// TwinCAT 3 PLC project HAWino
// ProgramVersion: 3.1.4024.12
// libraries:
//   Tc2_Standard, * (Beckhoff Automation GmbH)
//   Tc2_System, * (Beckhoff Automation GmbH)
//   Tc2_Utilities, * (Beckhoff Automation GmbH)
//   Tc3_IotBase, * (Beckhoff Automation GmbH)
//   Tc3_JsonXml, * (Beckhoff Automation GmbH)
//   Tc3_Module, * (Beckhoff Automation GmbH)
// project tree:
//   / ControlTask.TcTTO, Kollisionserkennung_1.TcTTO, MQTT_1.TcTTO, PlcTask.TcTTO
//   DUTs/ Auftrag.TcDUT, ControllerState.TcDUT, CoreDriveState.TcDUT, CoreGripperControlState.TcDUT, RobotInternalData.TcDUT, RobotPoseSimple.TcDUT, RobotStatusGW1.TcDUT, U_IpAdr.TcDUT, RobotPose.TcDUT
//   DUTs/PowerManagement/ FleetManagement.TcDUT, ST_PwrMgmt_HAWino.TcDUT, ST_PwrMgmt_HAWino_In.TcDUT, ST_PwrMgmt_HAWino_Out.TcDUT
//   DUTs/Sys/ DUT_SysState.TcDUT
//   GVLs/ ControlParameters.TcGVL, Var_HAWIno.TcGVL
//   POUs/HAWinoCore/ Camera.TcPOU, CameraConnectionUDP.TcPOU, Gripper.TcPOU, IrDistanceFromRaw.TcPOU, IrDistanceSensors.TcPOU, MotorDrivers.TcPOU, MQTT.TcPOU, PowerManager.TcPOU, WheelEncoders.TcPOU, HAWino.TcPOU
//   POUs/UserPOUs/GW2/ AStar.TcPOU, DS_GW1.TcPOU, Fahrauftrag.TcPOU, Kollisionserkennung.TcPOU, ReadAssigment.TcPOU
//   POUs/UserPOUs/GW3ControlAlgorithm/ CollisionDetector.TcPOU, KalmanObserver.TcPOU, NonLinearController.TcPOU, Robot.TcPOU, SimpleObserver.TcPOU, PController.TcPOU, SimpleTrajectory.TcPOU, TimeOptimalTrajectory.TcPOU, ControlPRG.TcPOU, VelocityMeasurement.TcPOU
//   POUs/UserPOUs/ FKT_Scale.TcPOU, TrajectoryControl.TcPOU
//   POUs/UserPOUs/GW3PathAndTrajectoryPlanning/ BezierCurve.TcPOU, LinearCurve.TcPOU, Path.TcPOU, Curve.TcPOU, TrajectoryPlanner.TcPOU
//   POUs/UserPOUs/UserFunctions/ AddMat3.TcPOU, AddRPS.TcPOU, ArrayToStruct.TcPOU, ATAN2.TcPOU, calcTimeDiff.TcPOU, FILL.TcPOU, MatDet3.TcPOU, MatInv3.TcPOU, MatrixTimesRPS.TcPOU, MatTimesMat.TcPOU, MatTimesRPS.TcPOU, normalizeAngle.TcPOU, Robot2World.TcPOU, RPS2RP.TcPOU, RPS2ARRAY.TcPOU, RP2ARRAY.TcPOU, ScaleRPS.TcPOU, shiftCamAngle.TcPOU, SI.TcPOU, SubstractMat3.TcPOU, SubtractRPS.TcPOU, ToRobotPoseSimple.TcPOU, World2Robot.TcPOU, ZEROS.TcPOU, ZEROS_INT.TcPOU, ZEROS_RobotPoseSimple.TcPOU
// real-time tasks:
//   TASK PlcTask: cycle T#10ms, priority 25, ADS port 350
//   TASK MQTT: cycle T#100000us, priority 11, ADS port 351
//   TASK TcCOM_DataAquisition: cycle T#10ms, priority 4, ADS port 352
//   TASK TcCOM_DataProcessing: cycle T#10ms, priority 14, ADS port 353
//   TASK ControlTask: cycle T#2ms, priority 1, ADS port 354
//   TASK A_search: cycle T#20ms, priority 22, ADS port 355
//   TASK Kollisionserkennung_1: cycle T#10ms, priority 21, ADS port 356
// I/O:
//   DEVICE Gerät 1 (EtherCAT), AmsNetId 192.168.1.44.2.1
//     Klemme 1 (EK1200) [EK1200-5000 EtherCAT Netzteil (2A E-Bus)]
//       Motorklemme A2 (EL7342) [EL7342 2K. DC-Motor-Endstufe (50V, 3.5A)]
//       Motorklemme A3 (EL7342) [EL7342 2K. DC-Motor-Endstufe (50V, 3.5A)]
//       Digitale Eingänge A4 (EL1008) [EL1008 8K. Dig. Eingang 24V, 3ms]
//       Digitale Ausgänge A5 (EL2004) [EL2004 4K. Dig. Ausgang 24V, 0.5A]
//       Analoge Eingänge A6 (EL3068) [EL3068 8K. Ana. Eingang 0-10V]
//       Analoge Eingänge A7 (EL3104) [EL3104 4K. Ana. Eingang +/-10V Diff.]
//       Temperaturklemme A8 (EL3204) [EL3204 4K. Ana. Eingang PT100 (RTD)]
//       Klemme 9 (EL9011) [EL9011 Endklemme]
//   DEVICE Gerät 2 (RT-Ethernet Adapter)
// variable links:
//   HAWino/HAWino Instance <-> Device 1 (EtherCAT)/Term 1 (EK1200)/Analoge Eingänge A6 (EL3068)
//     PlcTask Inputs/IrDistanceSensors.distanceRaw[{1..8}] <-> AI Standard Channel {1..8}/Value  (8 links)
//   HAWino/HAWino Instance <-> Device 1 (EtherCAT)/Term 1 (EK1200)/Analoge Eingänge A7 (EL3104)
//     PlcTask Inputs/IrDistanceSensors.distanceRaw[9] <-> AI Standard Channel 1/Value
//     PlcTask Inputs/PowerManager.batteryVoltageRaw <-> AI Standard Channel 3/Value
//     PlcTask Inputs/PowerManager.supplyCurrentRaw <-> AI Standard Channel 2/Value
//   HAWino/HAWino Instance <-> Device 1 (EtherCAT)/Term 1 (EK1200)/Digitale Ausgänge A5 (EL2004)
//     PlcTask Outputs/PowerManager.shutdownTrigger <-> InitiateShutdown/Output
//   HAWino/HAWino Instance <-> Device 1 (EtherCAT)/Term 1 (EK1200)/Digitale Eingänge A4 (EL1008)
//     ControlTask Inputs/ControlPRG.robot.bumper <-> Bumper (S1)/Input
//     ControlTask Inputs/ControlPRG.robot.slider <-> Channel 5/Input
//     ControlTask Inputs/MotorDrivers.bumper <-> Channel 3/Input
//     PlcTask Inputs/Gripper.partGripped <-> Channel 6/Input
//     PlcTask Inputs/PowerManager.shutdownButton <-> ShutdownRequested (S11)/Input
//   HAWino/HAWino Instance <-> Device 1 (EtherCAT)/Term 1 (EK1200)/Motorklemme A2 (EL7342)
//     ControlTask Inputs/ControlPRG.robot.vel.n1MotorRaw <-> DCM Synchron info data Channel 1/Info data 1
//     ControlTask Inputs/ControlPRG.robot.vel.n2MotorRaw <-> DCM Synchron info data Channel 2/Info data 1
//     ControlTask Inputs/WheelEncoders.encDataFromMotor1 <-> ENC Status compact Channel 1/Counter value
//     ControlTask Inputs/WheelEncoders.encDataFromMotor2 <-> ENC Status compact Channel 2/Counter value
//     ControlTask Outputs/MotorDrivers.enableToMotor1 <-> DCM Control Channel 1/Control/Enable
//     ControlTask Outputs/MotorDrivers.enableToMotor2 <-> DCM Control Channel 2/Control/Enable
//     ControlTask Outputs/MotorDrivers.velocityToMotor1 <-> DCM Velocity Channel 1/Velocity
//     ControlTask Outputs/MotorDrivers.velocityToMotor2 <-> DCM Velocity Channel 2/Velocity
//   HAWino/HAWino Instance <-> Device 1 (EtherCAT)/Term 1 (EK1200)/Motorklemme A3 (EL7342)
//     ControlTask Inputs/ControlPRG.robot.vel.n3MotorRaw <-> DCM Synchron info data Channel 1/Info data 1
//     ControlTask Inputs/WheelEncoders.encDataFromMotor3 <-> ENC Status compact Channel 1/Counter value
//     ControlTask Outputs/MotorDrivers.enableToMotor3 <-> DCM Control Channel 1/Control/Enable
//     ControlTask Outputs/MotorDrivers.velocityToMotor3 <-> DCM Velocity Channel 1/Velocity
//     PlcTask Outputs/Gripper.driveEnable <-> DCM Control Channel 2/Control/Enable
//     PlcTask Outputs/Gripper.driveVelocity <-> DCM Velocity Channel 2/Velocity
//   HAWino/HAWino Instance <-> Device 1 (EtherCAT)/Term 1 (EK1200)/Temperaturklemme A8 (EL3204)
//     MQTT_1 Inputs/MQTT.nBatteryTemperature <-> RTD Inputs Channel 1/Batterytemperature
//   HAWino/HAWino Instance <-> HAWino/HAWino Instance
//     ControlTask Inputs/ControlPRG.newWaypointListAvailable <-> PlcTask Outputs/Fahrauftrag.TrajectoryController.newWaypointListAvailable
//     ControlTask Inputs/ControlPRG.robotPoses <-> PlcTask Outputs/Camera.cameraData.robotPosition
//     ControlTask Inputs/ControlPRG.waypointList <-> PlcTask Outputs/Fahrauftrag.TrajectoryController.waypointList
//     ControlTask Inputs/ControlPRG.xBoEnable <-> PlcTask Outputs/Fahrauftrag.TrajectoryController.xBoEnable
//     ControlTask Inputs/ControlPRG.xBoReset <-> PlcTask Outputs/Fahrauftrag.TrajectoryController.xBoReset
//     ControlTask Inputs/MotorDrivers.vThetaCartesianToMotors <-> ControlTask Outputs/ControlPRG.robot.vThetaToRobot
//     ControlTask Inputs/MotorDrivers.vXCartesianToMotors <-> ControlTask Outputs/ControlPRG.robot.vXtoRobot
//     ControlTask Inputs/MotorDrivers.vYCartesianToMotors <-> ControlTask Outputs/ControlPRG.robot.vYtoRobot
//     Kollisionserkennung_1 Inputs/Kollisionserkennung.robotPoseArray <-> PlcTask Outputs/Camera.cameraData.robotPosition
//     Kollisionserkennung_1 Inputs/Kollisionserkennung.vxRobot <-> ControlTask Outputs/ControlPRG.robot.vXtoRobot
//     Kollisionserkennung_1 Inputs/Kollisionserkennung.vyRobot <-> ControlTask Outputs/ControlPRG.robot.vYtoRobot
//     MQTT_1 Inputs/MQTT.FeedbackToGW1 <-> PlcTask Outputs/Fahrauftrag.FeedbackToGW1
//     MQTT_1 Inputs/MQTT.RoboNmbToGoBack <-> PlcTask Outputs/Fahrauftrag.RoboNmbToGoBack
//     MQTT_1 Inputs/MQTT.resetGoBack <-> PlcTask Outputs/Fahrauftrag.resetGoBack
//     MQTT_1 Inputs/MQTT.resetVar <-> PlcTask Outputs/Fahrauftrag.resetVarMQTT
//     MQTT_1 Inputs/MQTT.stMqtt_HAWino_In/bComCheckAnswer <-> MQTT_1 Outputs/MQTT.bComCheckAnswer
//     MQTT_1 Inputs/MQTT.stMqtt_HAWino_In/nRobotNumber <-> PlcTask Outputs/HAWino.Robot_Number
//     MQTT_1 Inputs/MQTT.txtReadInit <-> PlcTask Outputs/HAWino.initDone
//     PlcTask Inputs/Fahrauftrag.Auftrag <-> MQTT_1 Outputs/MQTT.Auftrag
//     PlcTask Inputs/Fahrauftrag.StatusFromGW1 <-> MQTT_1 Outputs/MQTT.StatusFromGW1
//     PlcTask Inputs/Fahrauftrag.TrajectoryController.yBoArrivedAtDestination <-> ControlTask Outputs/ControlPRG.yBoArrivedAtDestination
//     PlcTask Inputs/Fahrauftrag.TrajectoryController.yControllerState <-> ControlTask Outputs/ControlPRG.state
//     PlcTask Inputs/Fahrauftrag.TrajectoryController.yRPposition <-> ControlTask Outputs/ControlPRG.yRPposition
//     PlcTask Inputs/Fahrauftrag.TrajectoryController.yUintWaypointIndex <-> ControlTask Outputs/ControlPRG.yUintWaypointIndex
//     PlcTask Inputs/Fahrauftrag.TrajectoryController.yVworldRef <-> ControlTask Outputs/ControlPRG.yVworldRef
//     PlcTask Inputs/Fahrauftrag.collision <-> ControlTask Outputs/ControlPRG.collision
//     PlcTask Inputs/Fahrauftrag.goBack <-> MQTT_1 Outputs/MQTT.goBack
//     PlcTask Inputs/Fahrauftrag.reset <-> MQTT_1 Outputs/MQTT.resetButton
//     PlcTask Inputs/Gripper.closeGripperCommand <-> PlcTask Outputs/Fahrauftrag.closeGripperCommand
//   HAWino/HAWino Instance <-> TcCOM Objects/Object2 (SoC_Model_Data_Aquisition_2022)
//     PlcTask Outputs/PowerManager.stMqtt_HAWino_IN/fActualBatteryCurrent <-> SoC_Model_Data_Aquisition_202_U/Current
//     PlcTask Outputs/PowerManager.stMqtt_HAWino_IN/fActualBatteryVoltage <-> SoC_Model_Data_Aquisition_202_U/Voltage
//   HAWino/HAWino Instance <-> TcCOM Objects/Object2 (SoC_Model__Data_Processing_2022)
//     MQTT_1 Inputs/MQTT.stMqtt_HAWino_In/bCheckCurrentDetected <-> SoC_Model__Data_Processing_20_Y/CACCheckDetected
//     MQTT_1 Inputs/MQTT.stMqtt_HAWino_In/fActualBatteryCurrent <-> SoC_Model__Data_Processing_20_Y/CurrentOut
//     MQTT_1 Inputs/MQTT.stMqtt_HAWino_In/fActualBatteryVoltage <-> SoC_Model__Data_Processing_20_Y/VoltageOut
//     MQTT_1 Inputs/MQTT.stMqtt_HAWino_In/fSoC <-> SoC_Model__Data_Processing_20_Y/SoC
//     MQTT_1 Inputs/MQTT.stMqtt_HAWino_In/nEstimatedChargingTime <-> SoC_Model__Data_Processing_20_Y/EstimatedChargingTime
//     MQTT_1 Inputs/MQTT.stMqtt_HAWino_In/nEstimatedRunningTime <-> SoC_Model__Data_Processing_20_Y/EstimatedRunningTime
//   TcCOM Objects/Object2 (SoC_Model_Data_Aquisition_2022) <-> TcCOM Objects/Object2 (SoC_Model__Data_Processing_2022)
//     SoC_Model_Data_Aquisition_202_Y/Coulombs <-> SoC_Model__Data_Processing_20_U/Coulombs
//     SoC_Model_Data_Aquisition_202_Y/CurrentMean <-> SoC_Model__Data_Processing_20_U/Current
//     SoC_Model_Data_Aquisition_202_Y/VoltageMean <-> SoC_Model__Data_Processing_20_U/Voltage

CONFIGURATION HAWino
    RESOURCE PLC ON TwinCAT3
        TASK ControlTask(INTERVAL := T#2ms, PRIORITY := 23);
        TASK Kollisionserkennung_1(INTERVAL := T#10ms, PRIORITY := 21);
        TASK MQTT_1(INTERVAL := T#100000us, PRIORITY := 11);
        TASK PlcTask(INTERVAL := T#10ms, PRIORITY := 25);
        PROGRAM MotorDrivers WITH ControlTask : MotorDrivers;
        PROGRAM WheelEncoders WITH ControlTask : WheelEncoders;
        PROGRAM ControlPRG WITH ControlTask : ControlPRG;
        PROGRAM Kollisionserkennung WITH Kollisionserkennung_1 : Kollisionserkennung;
        PROGRAM MQTT WITH MQTT_1 : MQTT;
        PROGRAM HAWino WITH PlcTask : HAWino;
        PROGRAM Fahrauftrag WITH PlcTask : Fahrauftrag;
    END_RESOURCE
END_CONFIGURATION

// ---- DUTs/Auftrag.TcDUT
TYPE Auftrag : //Fahrtauftrag
STRUCT
	Art: STRING;					//Fahrtauftag oder Ladeauftrag
	AbholStation : INT;				//Station 1...4, wo Teil aktuell liegt
	AbholTasche : INT;				//Tasche 1...4, wo Teil aktuell liegt
	AblageStation: INT;				//Station 1...4, wo Teil hinsoll
	AblageTasche : INT;				//Tasche 1...4, wo Teil hinsoll
END_STRUCT
END_TYPE

// ---- DUTs/ControllerState.TcDUT
{attribute 'qualified_only'}
{attribute 'strict'}
TYPE ControllerState :
(
	init 			:= 0,
	idle			:= 1,
	calcTrajectory 	:= 2,
	setTrajectory	:= 3,
	ready			:= 4,
	driving			:= 5,
	error			:= 6

);
END_TYPE

// ---- DUTs/CoreDriveState.TcDUT
{attribute 'qualified_only'}
{attribute 'strict'}
TYPE CoreDriveState :
(
	Init,
	Drive,
	BumperStop
);
END_TYPE

// ---- DUTs/CoreGripperControlState.TcDUT
{attribute 'qualified_only'}
{attribute 'strict'}
TYPE CoreGripperControlState :
(
	Open,
	Closing,
	Closed,
	Opening
);
END_TYPE

// ---- DUTs/PowerManagement/FleetManagement.TcDUT
TYPE FleetManagement :
STRUCT
	
	nRobotNumber			: INT;
	fSoC					: LREAL;
	nEstimatedRunningTime	: UDINT;
	ChargeRequired			: BOOL;
	
END_STRUCT
END_TYPE

// ---- DUTs/PowerManagement/ST_PwrMgmt_HAWino.TcDUT
TYPE ST_PwrMgmt_HAWino :
STRUCT
	Output	: ST_PwrMgmt_HAWino_In;		// Im Vergleich zur Chargingstation_3 sind hier Input und Output vertauscht!
	Input	: ST_PwrMgmt_HAWino_Out;
END_STRUCT
END_TYPE

// ---- DUTs/PowerManagement/ST_PwrMgmt_HAWino_In.TcDUT
TYPE ST_PwrMgmt_HAWino_In :
STRUCT
	nRobotNumber			: INT;
	tTimestamp				: TIME;		// The smallest unit of time is one millisecond. Example: T#82m47s295ms
	fSoC					: LREAL;
	fActualBatteryCurrent	: LREAL;
	fActualBatteryVoltage	: LREAL;
	fBatteryTemperature		: LREAL;
	nEstimatedRunningTime	: UDINT;	
	nEstimatedChargingTime	: UDINT;	
	bCheckCurrentDetected	: BOOL;		// 1. Bezeichnung: bNoChargingCurrent
	bComCheckAnswer			: BOOL;		// HAWino answer for communication check
END_STRUCT
END_TYPE

// ---- DUTs/PowerManagement/ST_PwrMgmt_HAWino_Out.TcDUT
TYPE ST_PwrMgmt_HAWino_Out :
STRUCT
	bChargingActive					: BOOL;
	bExternalRecalibrationTrigger	: BOOL;
	fExternalRecalibrationValue		: LREAL;
	bComCheckRequest 				: BOOL;		// Request from charger to HAWino to test stable communication 
END_STRUCT 
END_TYPE

// ---- DUTs/RobotInternalData.TcDUT
TYPE RobotInternalData :
	STRUCT
		Robot_Number : INT;
		Robot_IP_WiFi     : T_AmsNetId;
		Robot_IP_Wire     : T_AmsNetId;
		Robot_Name     : STRING;
		Robot_Nickname : STRING;
	END_STRUCT
END_TYPE

// ---- DUTs/RobotPoseSimple.TcDUT
TYPE RobotPoseSimple:
STRUCT
	x, y, theta : LREAL;
END_STRUCT
END_TYPE

// ---- DUTs/RobotStatusGW1.TcDUT
TYPE RobotStatusGW1 :
STRUCT
	Status : STRING;
END_STRUCT
END_TYPE

// ---- DUTs/Sys/DUT_SysState.TcDUT
{attribute 'qualified_only'}
{attribute 'strict'}
TYPE DUT_SysState :
(
	init:=0,
	preOp:=1,
	Op := 2,
	Error:=3
);
END_TYPE

// ---- DUTs/U_IpAdr.TcDUT
TYPE U_IpAdr :
UNION
	ipAdrInternal : UDINT;
	ipAdr : ARRAY[0..3] OF BYTE;
END_UNION
END_TYPE

// ---- DUTs/RobotPose.TcDUT
TYPE RobotPose EXTENDS RobotPoseSimple: 
STRUCT
	e : LREAL;
END_STRUCT
END_TYPE

// ---- GVLs/ControlParameters.TcGVL
{attribute 'qualified_only'}
VAR_GLOBAL

	//+++++++++++++++++++++++++++++++++++++++++++++++++++	
	//Parameters for ControlPRG
	//+++++++++++++++++++++++++++++++++++++++++++++++++++
	
	FeedForwardLinearization: BOOL := FALSE;

	//+++++++++++++++++++++++++++++++++++++++++++++++++++	
	//Parameters for PController (Controller)
	//+++++++++++++++++++++++++++++++++++++++++++++++++++
	
	//controller Gain Matrix
	controllerK: ARRAY [0..2,0..2] OF LREAL := [4,0,0,
									  0,4,0,
									  0,0,0.5];
									  
	//Maximal Translational Velocity (vX, vY)
	vtrans_max: LREAL := 934;
	//Maximal rotational Velocity (vTheta)
	vrot_max: LREAL   := 6.9;
	
	// accuracy tolerance
	accuracyXY: LREAL := 3;
	accuracyTheta: LREAL := 0.01;
	
					
	//+++++++++++++++++++++++++++++++++++++++++++++++++++	
	//Parameters for KalmanObserver (Observer)
	//+++++++++++++++++++++++++++++++++++++++++++++++++++
	
	//amount of cycles camera is delayed (Camdelay 123ms / Cycletyme 2ms)
	kObsDelayedCycles: INT	:= 61;
	
	//Encoder Process Noise Covariance Matrix
	Q : ARRAY [0..2,0..2] OF LREAL 		:=[9.3047,    0.4415,   -0.0036,
    									   0.4415,    26.0708,   -0.0078,
   										  -0.0036,   -0.0078,    0.0007];
	//Camera Measurement Covariance Matrix								  
	RMat : ARRAY [0..2, 0..2] OF LREAL 	:= [0.00127820524383046,    -0.00144745069148629,    1.57202639633006E-06,
											-0.00144745069148629,    0.0142936660651043,      -2.43008878392535E-05,
											1.57202639633006E-06,    -2.43008878392535E-05,	  2.50703907504212E-07];
	
													
	//+++++++++++++++++++++++++++++++++++++++++++++++++++	
	//Parameters for TimeOptimalTrajectory
	//+++++++++++++++++++++++++++++++++++++++++++++++++++
	
	//!!! IMPORTANT: Parameters in m not mm!!!
	
	// Bezier radius												
    maxRadius		    : LREAL				:= 0.1;
	
	samplingTime		: LREAL				:= 0.05;
	
	
	maxVel				: LREAL				:= 0.6;
	maxAcc				: LREAL				:= 0.5;
	
	arcLengthSlow		: LREAL				:= 0.22;
	maxSlowVel			: LREAL				:= 0.08;
	
	maxRotVel			: LREAL				:= 100;
	maxRotAcc			: LREAL				:= 100;	
	
	thetaDZ				: LREAL				:= 0.1;
	
END_VAR

// ---- GVLs/Var_HAWIno.TcGVL
{attribute 'qualified_only'}

// Roboternummern:
// 
// CX-31C9D6 = 1
// CX-35CFB8 = 2
// CX-35CDC8 = 3 	!!Vorläufig
// CX-35CDD6 = 4
// CX-4D0046 = 5

VAR_GLOBAL
	Robot_Number 				: INT :=2;
	CONTROLLER_CYCLE_TIME	 	: LREAL := 2E-3; //==> manual adjustment in SimpleObserverST required
END_VAR

// ---- POUs/HAWinoCore/MotorDrivers.TcPOU
PROGRAM MotorDrivers
VAR	
	//Zustandsautomat
	state:		CoreDriveState	:=	CoreDriveState.init;

	//Achsen Freischalten
	enableMotors: BOOL	:=0;

	//Umgerechnete Werte
	vX:		LREAL:=0;
	vY:		LREAL:=0;
	vTheta:	LREAL:=0;

	//Fahrrichtung Motor
	velocityMotor1 :LREAL:=0;
	velocityMotor2 :LREAL:=0;
	velocityMotor3 :LREAL:=0;
	
	//Skalierung auf MaxGeschwindigkeit Skalierung hängt mit CoE Register 8020:07 8020:08 zusammen !!!
	velocityMax:LREAL:=942.4777961;// Nenndrehzahl U/min CoE Register 8020:07 8020:08 fesgelegt Faktor 16 Wegen Getriebe 1:16
	velocityMotorsTf:LREAL:=0;
	
	// Skalierung auf Ansteuersignale LREAL=>WORD   Skalierung hängt mit CoE Register 8020:07 8020:08 zusammen !!!
	skalPos:LREAL:=34.7668668;//  MaxValue/MaxVelocity   [1/ mm/s]   32767/(942mm/s)   MaxVelocity=D*PI*n/(16*60) //16:1 Getriebeübersetzung  
	skalNeg:LREAL:=34.76792783;//  MaxVelau/MaxVelocity   [1/ mm/s]   32768/(942mm/s)   MaxVelocity=(80mm*PI*3600 U/min)/(16*60sec/min)
	
	//Inputs: CartesianToMotors + Bumper
	vXCartesianToMotors 	AT%I*:	LREAL:=0;
	vYCartesianToMotors 	AT%I*:	LREAL:=0;
	vThetaCartesianToMotors AT%I*:	LREAL:=0;
	bumper	   				AT%I*:	BOOL:=0;
	bumperStopReset 		AT%I*: 	BOOL:=0;
	
	//Outputs: Motor Values and Enable Signal
	enableToMotor1 AT%Q*:BOOL:=FALSE;
	enableToMotor2 AT%Q*:BOOL:=FALSE;
	enableToMotor3 AT%Q*:BOOL:=FALSE;
	
	velocityToMotor1 AT%Q*:INT:=0;
	velocityToMotor2 AT%Q*:INT:=0;
	velocityToMotor3 AT%Q*:INT:=0;
	
	counter: ULINT;
	Test: LREAL;
END_VAR
VAR CONSTANT
	Revisionsnummer: REAL:=0.3;// Vor dem Hochladen Nummer inkrementieren. Dadurch lässt sich prüfen, ob die neuste Version online ist.
END_VAR


(****** Konverzierung ToMotors Anfang************
Übersetzung der Koordinatentransformation aus dem Simulink Starterkit

	  conversion from positive and / or negative longitudinal, lateral and
	  rotational velocities(in milimeters per second) to three separate
	  positive motor velocities(resolution: 1Byte) and their rotation direction
inputs:  	vX  (longitudinal velocity in milimeters per second)
         	vY  (lateral velocity in milimeters per second)
			vTheta     (rotational velocity in milimeters per second)
outputs : velocityToMotor1	
			velocityToMotor2
			velocityToMotor3
conversion from longitudinal, lateral & rotational velocity to the
three separate motor velocities
*)


vX:=-vXCartesianToMotors;
vY:=-vYCartesianToMotors;
vTheta:=-vThetaCartesianToMotors;
Test:=EXPT(2,-1024);
velocityMotor1 := (-vX * COS(30.0*PI/180))	+ (vY * COS(60.0*PI/180))	+ (vTheta * 135.0);
velocityMotor2 := 0.0						+ (-vY)						+ (vTheta * 135.0);
velocityMotor3 := (vX * COS(30.0*PI/180))	+ (vY * COS(60.0*PI/180))	+ (vTheta * 135.0);

(* 	Geschwindigkeitsbegrenzung:
	Der Simulink Regler hat keine Output Begrenzung!
	Wenn Geschwindigkeit > v_max, dann muss v skaliert werden -> andere Motorgeschwindigkeiten müssen 
	dann entsprechend mitskaliert werden
	velocityMotorsTf: Faktor, der alle Geschwindigkeit auf v_max runterskaliert
*)
IF (velocityMotor1 > velocityMax) OR (velocityMotor1 < -velocityMax) THEN
    velocityMotorsTf:= velocityMotor1;
    IF (velocityMotorsTf = 0) THEN
			velocityMotorsTf:=1;
	END_IF
	// sign(velocityMotorsTf/ABS(velocityMotorsTf) = velocityMotorsTf/ABS(velocityMotorsTf)
    velocityMotor1:= velocityMotorsTf/ABS(velocityMotorsTf)*velocityMax;
    velocityMotor2:= velocityMotorsTf/ABS(velocityMotorsTf)*velocityMax/velocityMotorsTf * velocityMotor2 ;
    velocityMotor3:= velocityMotorsTf/ABS(velocityMotorsTf)*velocityMax/velocityMotorsTf * velocityMotor3 ;
END_IF

IF (velocityMotor2 > velocityMax) OR (velocityMotor2 < -velocityMax) THEN
    velocityMotorsTf:= velocityToMotor2;
    IF (velocityMotorsTf = 0) THEN
		velocityMotorsTf:=1;
	END_IF
	// sign(velocityMotorsTf/ABS(velocityMotorsTf) = velocityMotorsTf/ABS(velocityMotorsTf)
    velocityMotor1:= velocityMotorsTf/ABS(velocityMotorsTf)*velocityMax/velocityMotorsTf * velocityToMotor1;
    velocityMotor2:= velocityMotorsTf/ABS(velocityMotorsTf)*velocityMax;
    velocityMotor3:= velocityMotorsTf/ABS(velocityMotorsTf)*velocityMax/velocityMotorsTf * velocityToMotor3;
END_IF

IF (velocityMotor3 > velocityMax) OR (velocityMotor3 < -velocityMax) THEN
    velocityMotorsTf:= velocityToMotor3;
    IF (velocityMotorsTf = 0) THEN
			velocityMotorsTf:=1;
	END_IF
	// sign(velocityMotorsTf/ABS(velocityMotorsTf) = velocityMotorsTf/ABS(velocityMotorsTf)
    velocityMotor1:= velocityMotorsTf/ABS(velocityMotorsTf)*velocityMax/velocityMotorsTf * velocityMotor1;
    velocityMotor2:= velocityMotorsTf/ABS(velocityMotorsTf)*velocityMax/velocityMotorsTf * velocityMotor2 ;
    velocityMotor3:= velocityMotorsTf/ABS(velocityMotorsTf)*velocityMax;
END_IF
// Konvertierung ToMotors ENDE********************************************************


//MOTORANSTEUERUNG Zustandsautomat
CASE state OF
	CoreDriveState.init:						
						IF NOT bumper AND NOT bumperStopReset THEN
							state:=CoreDriveState.drive;
						END_IF
						
	CoreDriveState.drive:
						IF velocityMotor1>=0 THEN
							velocityToMotor1:=LREAL_TO_INT(velocityMotor1*skalPos);
						ELSE
							velocityToMotor1:=LREAL_TO_INT(velocityMotor1*skalNeg);
						END_IF
						
						IF velocityMotor2>=0 THEN
							velocityToMotor2:=LREAL_TO_INT(velocityMotor2*skalPos);
						ELSE
							velocityToMotor2:=LREAL_TO_INT(velocityMotor2*skalNeg);
						END_IF
						
						IF velocityMotor3>=0 THEN
							velocityToMotor3:=LREAL_TO_INT(velocityMotor3*skalPos);
						ELSE
							velocityToMotor3:=LREAL_TO_INT(velocityMotor3*skalNeg); 
						END_IF
							
							enableToMotor1:=1;
							enableToMotor2:=1;
							enableToMotor3:=1;
							
						IF bumper=TRUE THEN
							state:=CoreDriveState.BumperStop;
						END_IF
						
	CoreDriveState.BumperStop:
						velocityToMotor1:=0;
						velocityToMotor2:=0;
						velocityToMotor3:=0;
						enableToMotor1:=0;
						enableToMotor2:=0;
						enableToMotor3:=0;
						
						IF NOT bumper AND bumperStopReset THEN
							state := CoreDriveState.Init;
						END_IF
	ELSE
		state:=CoreDriveState.init;
END_CASE

END_PROGRAM

// ---- POUs/HAWinoCore/WheelEncoders.TcPOU
PROGRAM WheelEncoders
VAR
zaehler : UINT := 0;

//ENC Daten Differenzieren für Geschwindigkeit
diffConst:LREAL := Var_HAWIno.CONTROLLER_CYCLE_TIME;//SECONDS
encDataOldMotor1:UINT:=0;
encDataOldMotor2:UINT:=0;
encDataOldMotor3:UINT:=0;

//Koordinatentransformation Weg
skalEnc:LREAL:=0.00766990393;

//Koordinatentransformation Geschwindigkeit
v1:LREAL:=0;
v2:LREAL:=0;
v3:LREAL:=0;
velocityFromMotor1:LREAL:=0;
velocityFromMotor2:LREAL:=0;
velocityFromMotor3:LREAL:=0;

//INPUTS
encDataFromMotor1 AT%I*  :UINT:=0;
encDataFromMotor2 AT%I*  :UINT:=0;
encDataFromMotor3 AT%I*  :UINT:=0;

diff1: INT := 0;
diff2: INT := 0;
diff3: INT := 0;

//OUTPUTS
vXCartesianFromMotors AT%Q*:LREAL:=0;
vYCartesianFromMotors AT%Q*:LREAL:=0;
vthetaCartesianFromMotors AT%Q*:LREAL:=0;
END_VAR

IF MotorDrivers.state = CoreDriveState.Init THEN
	encDataOldMotor1 := encDataFromMotor1;
	encDataOldMotor2 := encDataFromMotor2;
	encDataOldMotor3 := encDataFromMotor3;
END_IF

// Encoder Wegberechnung und Differenzierung für Geschwindigkeit
diff1:=UINT_TO_INT(encDataFromMotor1) - UINT_TO_INT(encDataOldMotor1);
IF diff1 >= 32767 OR diff1 <= -32767 THEN
	diff1 := 0;
	zaehler := zaehler + 1;
END_IF
diff2:=UINT_TO_INT(encDataFromMotor2) - UINT_TO_INT(encDataOldMotor2);
IF diff2 >= 32767 OR diff2 <= -32767 THEN
	diff2 := 0;
END_IF
diff3:=UINT_TO_INT(encDataFromMotor3) - UINT_TO_INT(encDataOldMotor3);
IF diff3 >= 32767 OR diff3 <= -32767 THEN
	diff3 := 0;
END_IF

velocityFromMotor1:=diff1/diffConst*skalEnc;
velocityFromMotor2:=diff2/diffConst*skalEnc;
velocityFromMotor3:=diff3/diffConst*skalEnc;

// Koordinatentransformation Geschwindigkeit
v1:=-velocityFromMotor1;
v2:=-velocityFromMotor2;
v3:=-velocityFromMotor3;

vXCartesianFromMotors:=(v3 - v1) / (2.0 * COS(30.0*PI/180));  //in mm / s
vYCartesianFromMotors:=(v1 - 2.0 * v2 + v3) / 3.0;            //in mm / s
vThetaCartesianFromMotors:=(v1 + v2 + v3) / (3.0 * 135.0);    //in rad / s

// Alte Encoderdaten speichern
encDataOldMotor1:=encDataFromMotor1;
encDataOldMotor2:=encDataFromMotor2;
encDataOldMotor3:=encDataFromMotor3;

END_PROGRAM

// ---- POUs/UserPOUs/GW3ControlAlgorithm/ControlPRG.TcPOU
//Tracking controller:
// Main handling of the control algorithm
// implements a state machine with states: init, idle, calcTrajectory, ready, driving
// links the different components of the control algorithm: control law, observer, trajectory, robot, camera... => Maybe more needed later e.g. filter 
// links to GW2 via the defined interface

PROGRAM ControlPRG
VAR_INPUT
END_VAR
VAR_OUTPUT
END_VAR
VAR
	//declare objects
	kobserver		  : KalmanObserver;
	collisionDetector : collisionDetector;
	controller		  : PController;			//Control law object
	trajectory		  : TimeOptimalTrajectory;			//Trajectory Object
	robot			  : Robot;							//link to physical I/O of roboter or simulation model of the roboter
	robotPoses 	 AT%I*: ARRAY [1..8] OF RobotPose;	    //input from camera
	
	state AT%Q*: ControllerState := ControllerState.init;//sets controller state
	
	CONTROL_ERROR_THRESH : LREAL := 5;
	
	FFLin: BOOL := ControlParameters.FeedForwardLinearization;
	thetaLin: LREAL;
	
	///////////////////////////////////////////////
	///////////// LINKS TO GW2  ///////////////////
	///////////////////////////////////////////////
	
	//inputs from GW2, uncomment and link when needed
	xBoEnable AT%I*: BOOL := FALSE;							// implemented, Freigabesignal für Fahrt, Roboter stoppt bei FALSE
	xBoReset  AT%I*: BOOL := FALSE;							// implemented, reset error state => idle
	waypointList AT%I*: ARRAY[0..100] OF RobotPoseSimple;	// implemented, Wegpunktliste mit Roboter-Posen in globalen Koordinaten (x, y, theta)
	newWaypointListAvailable AT%I*: BOOL := FALSE;			// implemented, Status-Bit zur Signalisierung einer neuen WP-Liste
	
	//outputs to GW2, uncomment and link when needed
	yBoArrivedAtDestination AT%Q*:	BOOL := FALSE;			// implemented, TRUE, wenn Ziel erreicht, Ziel entspricht letzten gültigen WP
	yUintWaypointIndex 	AT%Q*: INT  := 0;					// implemented, COUNTER zur Anzeige, des Indexes des nächstes WP
	yRPposition 		AT%Q*: RobotPoseSimple;				// implemented, aktuelle Roboterposition, für Simulationszwecke
	yVworldRef			AT%Q*: RobotPoseSimple;
	collision			AT%Q*: ARRAY [0..4] OF BOOL;
END_VAR

//robot disabled by default
robot.enable			:= FALSE;

//outputs to GW2
yRPposition 			:= kobserver.yObserverdPose;
yUintWaypointIndex 		:= trajectory.WPLidx;
yVworldRef				:= controller.xRobotvelRef;
collision				:= collisionDetector.collisionDetected;

//call controller state machine
stateMachine();

//Select FF or FB linearization
IF FFLin = TRUE THEN
	thetaLin := trajectory.referencePose.theta;
ELSE
	thetaLin := kobserver.yObserverdPose.theta;		
END_IF
//transform roboter velocities into world velocities and pass them to Simulink
Robot2World( 
	vx_robot 	:= robot.vX,
	vy_robot 	:= robot.vY,
	omega_robot := robot.vTheta,
	theta		:= thetaLin,
	vx_world 	=> collisionDetector.vX,
	vy_world  	=> collisionDetector.vY);
	
collisionDetector(
	rawRobotPoses 	:= robotPoses,
	observedPose 	:= kobserver.yObserverdPose);
	
//initilizing and linking of control algorithm individual components
//init observer
kobserver(xCameraPose 	:= shiftCamAngle(camData := robotPoses[Var_HAWIno.Robot_Number], path := trajectory.path),
		 //xCameraPose 	:= robotPoses[Var_HAWIno.Robot_Number],
		 xVxRobot    	:= robot.vX,						//link x-velocity with measured velocity
		 xVyRobot    	:= robot.vY,						//link y-velocity with measured velocity
		 xOmegaRobot    := robot.vTheta,
 		 //xVxToRobot		:= controller.vXrobot,
		 //xVyToRobot		:= controller.vYrobot,
		 //xOmegaToRobot	:= controller.omegaRobot,				//link theta-velocity with measured velocity
		 theta			:= thetaLin);	

						//Angle for IO-Lineariztion						 
//init controller and link to observer
controller(xRobotPose 		:= kobserver.yObserverdPose,			//pass controller the observerd roboter pose
		   xRobotPoseRef	:= trajectory.referencePose,
		   xRobotVelRef		:= trajectory.referenceVelocities,
		   enable			:= robot.enable);		//pass controller the reference position for the next cycle comming from the trajectory

//trajectory object
trajectory(
	drive 			:= robot.enable,
	currentPose 	:= kobserver.yObserverdPose,					//Current implementation needs observed pose for distance calculation, TODO: check if needed for final implemenation
	referencePose 	=> controller.xRobotPoseRef					//outputs reference pose to controller
);

//observer.xCameraPose 	:= shiftCamAngle(camData := robotPoses[Var_HAWIno.Robot_Number], path := trajectory.path);
//transform control inputs into robot coordinates and pass them to the robot
//pass enable signal to robot
World2Robot(
			vx_world := controller.vXrobot,						//controller outputs vXref in world coordinates
			vy_world := controller.vYrobot,						//controller outputs vYref in world coordinates
			omega_world := controller.omegaRobot,				//controller outputs vThetaRef in world coordinates
			theta := thetaLin,									//trajectory theta for I/O Lin => FB-Structure
			vx_robot => robot.vXref,							//vXref in robot coordinates are passed to robot as control output
			vy_robot => robot.vYref,							//vYref in robot coordinates are passed to robot as control output
			omega_robot => robot.vThetaRef,
);

// to do:
IF trajectory.finished AND controller.reachedReference THEN
	yBoArrivedAtDestination := TRUE;
END_IF

//needs to be called so that the velocities will be written to motor drives
robot();

METHOD calculateTrajectory : BOOL
VAR_INPUT
END_VAR
trajectory.setWaypointList(waypointList);
END_METHOD

METHOD checkForFailure : BOOL
VAR_INPUT
END_VAR
checkForFailure := robot.bumperGotTriggered OR trajectory.generationFailed;
END_METHOD

METHOD drive : BOOL
VAR_INPUT
END_VAR
robot.enable := TRUE;
END_METHOD

METHOD init : BOOL
VAR_INPUT
END_VAR
VAR
END_VAR
END_METHOD

METHOD reset : BOOL
VAR_INPUT
END_VAR
reset := trajectory.reset() AND controller.reset() AND kobserver.reset();
END_METHOD

METHOD stateMachine : BOOL
VAR_INPUT
END_VAR
//control algorithms state machine
CASE state OF
	ControllerState.init:
		//initilize objects and link them
		init();
		//go into idle
		state := ControllerState.idle;
	
	ControllerState.idle:
		//if new waypointlist available reset trajectory and go into set trajectory state
		IF checkForFailure() THEN
			state := ControllerState.error;
		ELSIF newWaypointListAvailable THEN
			IF reset() THEN
				state := ControllerState.setTrajectory;
			END_IF
		END_IF
	
	ControllerState.setTrajectory:
		//got new trajectory so not anymore at destination
		yBoArrivedAtDestination := FALSE;
		//calculate trajectory
		trajectory.setWaypointList(waypointList);
			
		//go into calcTrajectory as soon as GW2 resets the new waypointlist flag to avoid looping through
		//ready --> setTrajectory --> calcTrajectory
		IF checkForFailure() THEN
			state := ControllerState.error;	
		ELSIF NOT newWaypointListAvailable AND trajectory.pathReady THEN
			state := ControllerState.calcTrajectory;
		END_IF
		
	 ControllerState.calcTrajectory:
		trajectory.generateTrajectory();
	 	IF checkForFailure() THEN
			state := ControllerState.error;
		ELSIF trajectory.ready THEN
			state := ControllerState.ready;
		END_IF
		
	
	ControllerState.ready:
		IF newWaypointListAvailable THEN
			//stop and calculate new trajectory
			IF reset() THEN
				state := ControllerState.setTrajectory;
			END_IF
		ELSIF xBoEnable THEN
			state := ControllerState.driving;
		END_IF
	
	ControllerState.driving:
		
		IF checkForFailure() THEN
			state := ControllerState.error;
		ELSIF newWaypointListAvailable THEN
			//stop and calculate new trajectory
			IF reset() THEN
				state := ControllerState.setTrajectory;
			END_IF
		ELSIF yBoArrivedAtDestination OR robot.sliderGotTriggered THEN
			yBoArrivedAtDestination := TRUE; //only relevant if transition is triggered through the slider
			//got back to idle and set arrived flag for GW2, method needed?
			IF reset() THEN
				state := ControllerState.idle;
			END_IF
		ELSIF xBoEnable THEN
			//do the driving
			drive();
		ELSE
			//if xBoEnable isn't set anymore go into ready and wait for it again
			state := ControllerState.ready;
		END_IF
		
	ControllerState.error:
		IF xBoReset THEN
			reset();
			state := ControllerState.idle;
		END_IF
END_CASE
END_METHOD

END_PROGRAM

// ---- POUs/UserPOUs/GW3ControlAlgorithm/KalmanObserver.TcPOU
//KalmanObserver:
//Implements a kalman observer which assumes the camera position is the true position of the robot whenever camera data arrives. 
FUNCTION_BLOCK KalmanObserver
VAR_INPUT
	xCameraPose:	RobotPoseSimple;
	xVxRobot: 		LREAL;
	xVyRobot: 		LREAL;
	xOmegaRobot: 	LREAL;
	theta:			LREAL; //theta for I/O Lineraztion only explicitly Input for FF-Linearization
END_VAR

VAR_OUTPUT
	yObserverdPose: 	RobotPoseSimple;
END_VAR

VAR
	newCamDataArrived: BOOL;
	camDataOld, observerError, observedPosition, lastValidCamData, vWorld: RobotPoseSimple;
	pulseGenerator: TP;
	
	delayedCycles		AT%Q* 	: INT	:= ControlParameters.kObsDelayedCycles;	//Camdelay 160ms / Cycletyme 2ms
	delayedPosition: ARRAY [0..140] OF RobotPoseSimple;

											
	P, H, TEMP : ARRAY [0..2,0..2] OF LREAL;

	Q : ARRAY [0..2,0..2] OF LREAL 		:= ControlParameters.Q;
										  
	(*Q : ARRAY [0..2,0..2] OF LREAL 		:=[0.0145,    0.2583,   -0.1632,
    									   0.1352,    0.0092,    0.2404,
   										   -0.4028,   0.1352,    0.0001]; *)
											  
	RMat : ARRAY [0..2, 0..2] OF LREAL 	:= ControlParameters.RMat;
											
(*	RMat : ARRAY [0..2, 0..2] OF LREAL 	:= [0.0291,		0.6199,		-0.5602,
											0.6455,		0.0307,      0.2979,
											-0.0226,    -0.0317,	 0.0098]; *)
											
	C : ARRAY [0..2,0..2] OF LREAL 		:=[1, 0, 0,
    									   0, 1, 0,
   										   0, 0, 1];
	// TEST
	//systime : NT_GetTime;
	observedPositionAP: RobotPoseSimple;
	PAP: ARRAY [0..2, 0..2] OF LREAL;
END_VAR

//transform roboter velocities into world velocities and pass them to Simulink
Robot2World( 
	vx_robot 	:= xVxRobot,
	vy_robot 	:= xVyRobot,
	omega_robot := xOmegaRobot,
	theta		:= yObserverdPose.theta,
	vx_world 	=> vWorld.x,
	vy_world  	=> vWorld.y,
	omega_world => vWorld.theta);
	
CheckForNewCameraData();	//Schreibt direkt in Variable  "newCamDataArrived"

//systime(START:=newCamDataArrived);	// TEST

delayPosition();

// Step 1 Prediction
observedPositionAP := AddRPS(observedPosition, ScaleRPS(c := Var_HAWIno.CONTROLLER_CYCLE_TIME, vWorld));
PAP := AddMat3(P, Q);




//if cam data arrived correct
IF newCamDataArrived THEN
	//Step 2 Optimize H
	TEMP := AddMat3(PAP,RMat);
	TEMP := MatInv3(TEMP);
	H := MatTimesMat(PAP, TEMP);
	
	//step 3 Correction
	//calculate observer error
	observerError := SubtractRPS(xCameraPose,delayedPosition[delayedCycles]);
	//correct observed position
	observedPosition := AddRPS(observedPositionAP, MatTimesRPS(H, observerError));
	//correct obersvation covariance
	P := SubstractMat3(PAP, MatTimesMat(H, PAP));
	lastValidCamData := xCameraPose;
ELSE 
	observedPosition := observedPositionAP;
	P := PAP;
END_IF


//set Outputs
yObserverdPose 	:= observedPosition;
camDataOld 		:= xCameraPose;

METHOD checkForNewCameraData : BOOL
VAR_INPUT
END_VAR
newCamDataArrived := (camDataOld.x <> xCameraPose.x OR camDataOld.y <> xCameraPose.y OR camDataOld.theta <> xCameraPose.theta) //cahnge in one of the positions
					 AND xCameraPose.x <> 0 AND xCameraPose.y <> 0;		//valid data
END_METHOD

METHOD PRIVATE delayPosition : BOOL
VAR_INPUT
END_VAR
VAR
	i: INT := 0;
END_VAR
FOR i := 0 TO delayedCycles-1 DO
	delayedPosition[i+1] := delayedPosition[i];
END_FOR
delayedPosition[0] := observedPosition;
END_METHOD

METHOD reset : BOOL
VAR_INPUT
END_VAR
VAR
	
END_VAR
reset := TRUE;
IF newCamDataArrived THEN
	observedPosition := xCameraPose;
ELSE
	observedPosition := lastValidCamData;
END_IF
END_METHOD

END_FUNCTION_BLOCK

// ---- POUs/UserPOUs/UserFunctions/Robot2World.TcPOU
//transformation of robot 2 world velocities
FUNCTION Robot2World 
VAR_INPUT
	vx_robot: 	 LREAL;
	vy_robot: 	 LREAL;
	omega_robot: LREAL;
	theta: 		 LREAL;
END_VAR

VAR_OUTPUT
	vx_world: 	 LREAL;
	vy_world: 	 LREAL;
	omega_world: LREAL;
END_VAR

VAR
END_VAR

vx_world 	:= COS(theta)*vx_robot - SIN(theta)*vy_robot;
vy_world 	:= SIN(theta)*vx_robot + COS(theta)*vy_robot;
omega_world := omega_robot;

END_FUNCTION

// ---- POUs/UserPOUs/UserFunctions/AddRPS.TcPOU
FUNCTION AddRPS : RobotPoseSimple
VAR_INPUT
	pose1, pose2: RobotPoseSimple;
END_VAR
VAR
END_VAR

AddRPS.x		:= pose1.x + pose2.x;
AddRPS.y		:= pose1.y + pose2.y;
AddRPS.theta	:= pose1.theta + pose2.theta;

END_FUNCTION

// ---- POUs/UserPOUs/UserFunctions/ScaleRPS.TcPOU
FUNCTION ScaleRPS : RobotPoseSimple
VAR_INPUT
	c: 		LREAL;
	pose: 	RobotPoseSimple;
END_VAR
VAR
END_VAR

ScaleRPS.x		:= c*pose.x;	
ScaleRPS.y		:= c*pose.y;
ScaleRPS.theta	:= c*pose.theta;

END_FUNCTION

// ---- POUs/UserPOUs/UserFunctions/AddMat3.TcPOU
FUNCTION AddMat3 : ARRAY[0..2, 0..2] OF LREAL
VAR_INPUT
	mat1: ARRAY[0..2, 0..2] OF LREAL;
	mat2: ARRAY[0..2, 0..2] OF LREAL;
END_VAR

VAR
	i, j: INT; 
END_VAR

FOR i := 0 TO 2 DO
	FOR j := 0 TO 2 DO
		AddMat3[i,j] := mat1[i,j] + mat2[i,j];
	END_FOR
END_FOR

END_FUNCTION

// ---- POUs/UserPOUs/UserFunctions/MatInv3.TcPOU
FUNCTION MatInv3 : ARRAY [0..2,0..2] OF LREAL
VAR_INPUT
	A : ARRAY [0..2,0..2] OF LREAL;
END_VAR

VAR
	det		: LREAL;
END_VAR

det := MatDet3(A);

MatInv3[0,0] := ( A[1,1]*A[2,2] - A[1,2]*A[2,1] ) / det;
MatInv3[0,1] := ( -A[0,1]*A[2,2] + A[0,2]*A[2,1] ) / det;
MatInv3[0,2] := ( A[0,1]*A[1,2] - A[0,2]*A[1,1] ) / det;
MatInv3[1,0] := ( -A[1,0]*A[2,2] + A[1,2]*A[2,0] ) / det;
MatInv3[1,1] := ( A[0,0]*A[2,2] - A[0,2]*A[2,0] ) / det;
MatInv3[1,2] := ( -A[0,0]*A[1,2] + A[0,2]*A[1,0] ) / det;
MatInv3[2,0] := ( A[1,0]*A[2,1] - A[1,1]*A[2,0] ) / det;
MatInv3[2,1] := ( -A[0,0]*A[2,1] + A[0,1]*A[2,0] ) / det;
MatInv3[2,2] := ( A[0,0]*A[1,1] - A[0,1]*A[1,0] ) / det;

END_FUNCTION

// ---- POUs/UserPOUs/UserFunctions/MatDet3.TcPOU
FUNCTION MatDet3 : LREAL
VAR_INPUT
	A : ARRAY [0..2,0..2] OF LREAL;
END_VAR

MatDet3 := A[0,0]*A[1,1]*A[2,2] + A[0,1]*A[1,2]*A[2,0] + A[0,2]*A[1,0]*A[2,1] - A[0,1]*A[1,0]*A[2,2] - A[0,2]*A[1,1]*A[2,0] - A[0,0]*A[1,2]*A[2,1];

END_FUNCTION

// ---- POUs/UserPOUs/UserFunctions/MatTimesMat.TcPOU
FUNCTION MatTimesMat : ARRAY [0..2,0..2] OF LREAL
VAR_INPUT
	A,B: ARRAY [0..2,0..2] OF LREAL;
END_VAR

MatTimesMat[0,0] := A[0,0]*B[0,0] + A[0,1]*B[1,0] + A[0,2]*B[2,0];
MatTimesMat[0,1] := A[0,0]*B[0,1] + A[0,1]*B[1,1] + A[0,2]*B[2,1];
MatTimesMat[0,2] := A[0,0]*B[0,2] + A[0,1]*B[1,2] + A[0,2]*B[2,2];
MatTimesMat[1,0] := A[1,0]*B[0,0] + A[1,1]*B[1,0] + A[1,2]*B[2,0];
MatTimesMat[1,1] := A[1,0]*B[0,1] + A[1,1]*B[1,1] + A[1,2]*B[2,1];
MatTimesMat[1,2] := A[1,0]*B[0,2] + A[1,1]*B[1,2] + A[1,2]*B[2,2];
MatTimesMat[2,0] := A[2,0]*B[0,0] + A[2,1]*B[1,0] + A[2,2]*B[2,0];
MatTimesMat[2,1] := A[2,0]*B[0,1] + A[2,1]*B[1,1] + A[2,2]*B[2,1];
MatTimesMat[2,2] := A[2,0]*B[0,2] + A[2,1]*B[1,2] + A[2,2]*B[2,2];

END_FUNCTION

// ---- POUs/UserPOUs/UserFunctions/SubtractRPS.TcPOU
FUNCTION SubtractRPS : RobotPoseSimple
VAR_INPUT
	pose1, pose2: RobotPoseSimple;
END_VAR
VAR
END_VAR

SubtractRPS.x		:= pose1.x - pose2.x;
SubtractRPS.y		:= pose1.y - pose2.y;
SubtractRPS.theta	:= pose1.theta - pose2.theta;

END_FUNCTION

// ---- POUs/UserPOUs/UserFunctions/MatTimesRPS.TcPOU
FUNCTION MatTimesRPS : RobotPoseSimple
VAR_INPUT
	K: ARRAY [0..2,0..2] OF LREAL;
	pose: RobotPoseSimple;
END_VAR

//2.) apply gain on errors
MatTimesRPS.x 	 := K[0,0] * pose.x + K[1,0] * pose.y + K[2,0] * pose.theta;
MatTimesRPS.y 	 := K[0,1] * pose.x + K[1,1] * pose.y + K[2,1] * pose.theta;
MatTimesRPS.theta := K[0,2] * pose.x + K[1,2] * pose.y + K[2,2] * pose.theta;

END_FUNCTION

// ---- POUs/UserPOUs/UserFunctions/SubstractMat3.TcPOU
FUNCTION SubstractMat3 : ARRAY[0..2, 0..2] OF LREAL
VAR_INPUT
	mat1: ARRAY[0..2, 0..2] OF LREAL;
	mat2: ARRAY[0..2, 0..2] OF LREAL;
END_VAR

VAR
	i, j: INT; 
END_VAR

FOR i := 0 TO 2 DO
	FOR j := 0 TO 2 DO
		SubstractMat3[i,j] := mat1[i,j] - mat2[i,j];
	END_FOR
END_FOR

END_FUNCTION

// ---- POUs/UserPOUs/GW3ControlAlgorithm/CollisionDetector.TcPOU
FUNCTION_BLOCK CollisionDetector
VAR_INPUT
	rawRobotPoses: 		ARRAY [1..8] OF RobotPose;
	observedPose: 						RobotPoseSimple;
	vX, vY:							    LREAL;
END_VAR
VAR_OUTPUT
	collisionDetected: 	ARRAY [0..4] OF BOOL;
END_VAR
VAR
	velocity: RobotPose;
	robotPoses, lastPoses, lastVelocities:				ARRAY [1..8] OF RobotPose;
	collsionCanditates:					ARRAY [0..4] OF BOOL; 			
	distance: 							LREAL;
	//Parameters
	nmbOfRobots:			 INT   := 4;
	boundBoxRadius:			 LREAL := 700;  //radius of Bounding Box
	collisionResetDistance:  LREAL := boundBoxRadius + 100; 
	
	cameraValid : ARRAY [0..4] OF BOOL;
	i : INT;
END_VAR

handleCameraData();
filterCollisionCandidates();
velocity.x := vX;
velocity.y := vY;

FOR i := 1 TO nmbOfRobots BY 1 DO	
	//only reset a detected collision if the distance between both robots is large enough
	IF i <> Var_HAWino.Robot_Number AND collisionDetected[i] THEN
		distance := SQRT(EXPT(robotPoses[i].x- rawRobotPoses[Var_HAWino.Robot_Number].x,2) + EXPT(robotPoses[i].y - rawRobotPoses[Var_HAWino.Robot_Number].y,2));
		IF distance > collisionResetDistance THEN
			collisionDetected[i] := FALSE;
			collisionDetected[Var_HAWino.Robot_Number] := FALSE;
		END_IF
	ELSIF i <> Var_HAWino.Robot_Number AND collsionCanditates[i] THEN
		distance := SQRT(EXPT(robotPoses[i].x- rawRobotPoses[Var_HAWino.Robot_Number].x,2) + EXPT(robotPoses[i].y - rawRobotPoses[Var_HAWino.Robot_Number].y,2));
		IF distance < boundBoxRadius THEN
			collisionDetected[i] := TRUE;
			collisionDetected[Var_HAWino.Robot_Number] := TRUE;
		END_IF
	END_IF
	

END_FOR

lastPoses := robotPoses;

METHOD filterCollisionCandidates 
VAR_INPUT
END_VAR
VAR
	phi, phiLower, phiUpper: LREAL;
	vxCandidate, vyCandidate, vAbsSelf, dVAbs, enclosedAngle, directionOfMovement: LREAL;	
	i : INT;
END_VAR
FOR i := 1 TO nmbOfRobots BY 1 DO
	//check for every Robot i wether it is moving toward this robot or if this robot is moving towards Robot i
	IF i <> Var_HAWino.Robot_Number THEN
		collsionCanditates[i]  := isCollisionPossible(candidateNmb := Var_HAWino.Robot_Number, targetNmb := i); //check if this HAWino is moving towards HAWino i
		collsionCanditates[i]  := isCollisionPossible(candidateNmb := i, targetNmb := Var_HAWino.Robot_Number); //check if this HAWino is moving towards HAWino i
	END_IF
END_FOR
END_METHOD

METHOD handleCameraData 
VAR_INPUT
END_VAR
VAR
	i : INT;
END_VAR
FOR i := 1 TO nmbOfRobots BY 1 DO
	cameraValid[i] := FALSE;
	IF i = Var_HAWIno.Robot_Number THEN //use observer data for the robot this fb is running on
		cameraValid[i] := TRUE;
		robotPoses[i] := RPS2RP(observedPose);
	ELSIF rawRobotPoses[i].x = robotPoses[i].x AND rawRobotPoses[i].y = robotPoses[i].y THEN
		cameraValid[i] := FALSE;
	ELSIF rawRobotPoses[i].x <> 0 AND rawRobotPoses[i].y <> 0 THEN //for all other robots only update robot pose if camera data is valid
		robotPoses[i] := rawRobotPoses[i];
		cameraValid[i] := TRUE;
	END_IF
END_FOR
END_METHOD

METHOD isCollisionPossible : BOOL
VAR_INPUT
	candidateNmb: 	INT;
	targetNmb:		INT;
END_VAR
VAR
	vxCandidate, vyCandidate: LREAL;
	directionOfMovement, directionOfTarget: LREAL;
END_VAR
//default
isCollisionPossible := FALSE;

//candidate can only collide if it is moving -> calculate velocities
IF candidateNmb <> Var_HAWino.Robot_Number AND cameraValid[candidateNmb] THEN
	//if candidate is not this robot -> differentiate cam data -> only if camera is valid otherwise v = 0
	vxCandidate  					:=  (robotPoses[candidateNmb].x - lastPoses[candidateNmb].x)/Var_HAWIno.CONTROLLER_CYCLE_TIME;	
	vyCandidate  					:=  (robotPoses[candidateNmb].y - lastPoses[candidateNmb].y)/Var_HAWIno.CONTROLLER_CYCLE_TIME;
	lastVelocities[candidateNmb].x  :=  vxCandidate;
	lastVelocities[candidateNmb].y  :=  vyCandidate;
ELSIF candidateNmb <> Var_HAWino.Robot_Number AND NOT cameraValid[candidateNmb] THEN
	//if camera is invalid then take the last known velocity
	vxCandidate := lastVelocities[candidateNmb].x;
	vyCandidate := lastVelocities[candidateNmb].y;
ELSE
	//if candidate is this robot -> take velocity measurements
	vxCandidate 		:= velocity.x;
	vyCandidate			:= velocity.y;
END_IF		

//if the candidate is moving
IF vxCandidate <> 0 OR vyCandidate <> 0 THEN
	//check in which direction it is moving
	directionOfMovement	:= ATAN2(y := vyCandidate, x:= vxCandidate);
	
	//check in which direction target robot is located
	directionOfTarget   := ATAN2(y := robotPoses[candidateNmb].y-robotPoses[targetNmb].y, x := robotPoses[candidateNmb].x-robotPoses[targetNmb].x);
	directionOfTarget 	:= normalizeAngle(angle := directionOfTarget, lowerBound := directionOfMovement - pi, upperBound := directionOfMovement + pi); //angle handling
	
	//potential collision if target is in the pi/2 bounding box of the movenent direction
	IF ABS(directionOfTarget-directionOfMovement) > pi/2 THEN
		isCollisionPossible := TRUE;
	END_IF
END_IF
END_METHOD

END_FUNCTION_BLOCK

// ---- POUs/UserPOUs/UserFunctions/RPS2RP.TcPOU
//Converts a RobotPoseSimple 2 RobotPose, assuming an error of 0
//NOTE: the reverse conversion is not needed because of polymorphmism of RobotPose, see Defintion of RobotPose STRUCT
FUNCTION RPS2RP : RobotPose
VAR_INPUT
	pose: RobotPoseSimple;
END_VAR
VAR
END_VAR

RPS2RP.x   		:= pose.x;
RPS2RP.y		:= pose.y;
RPS2RP.theta  	:= pose.theta;
RPS2RP.e		:= 0;

END_FUNCTION

// ---- POUs/UserPOUs/UserFunctions/ATAN2.TcPOU
FUNCTION ATAN2 : LREAL
VAR_INPUT
	y: LREAL;
	x: LREAL;
END_VAR
VAR
END_VAR

IF x > 0 THEN
	ATAN2 := ATAN(y/x);
ELSIF x < 0 AND y > 0 THEN
	ATAN2 :=  ATAN(y/x) + pi;
ELSIF x < 0 AND y = 0 THEN
	ATAN2 := pi;
ELSIF x < 0 AND y < 0 THEN
	ATAN2 := ATAN(y/x) - pi;
ELSIF x = 0 AND y > 0 THEN
	ATAN2 := pi/2;
ELSIF x = 0 AND y < 0 THEN
    ATAN2 := -pi/2;
END_IF

END_FUNCTION

// ---- POUs/UserPOUs/UserFunctions/normalizeAngle.TcPOU
FUNCTION normalizeAngle : LREAL
VAR_INPUT
	angle: 			LREAL;
	upperBound:		LREAL;
	lowerBound:		LREAL;
END_VAR
VAR
END_VAR

IF angle > upperBound THEN
	normalizeAngle := angle - 2*pi;
ELSIF angle < lowerBound THEN
	normalizeAngle := angle + 2*pi;
ELSE
	normalizeAngle := angle;
END_IF

END_FUNCTION

// ---- POUs/UserPOUs/GW3ControlAlgorithm/PController.TcPOU
(*PController:
Implements a simple state feedback law with a 3x3 control gain matrix 'K', 
a translation speed limit 'vtrans_max' (x- and y-axis) and a rotational speed 
limit 'vrot_max'.
*)
FUNCTION_BLOCK PController
VAR_INPUT
	xRobotPose: 		RobotPoseSimple; 				//current pose
	xRobotPoseRef: 		RobotPoseSimple; 				//reference pose
	xRobotvelRef: 		RobotPoseSimple;				//reference velocity
	enable:				BOOL 			:= FALSE;
END_VAR

VAR_OUTPUT
	//control outputs
	vXrobot:			LREAL;
	vYrobot:			LREAL;
	omegaRobot:			LREAL;
	reachedReference:	BOOL;
END_VAR

VAR
	//static control parameters
	K: ARRAY [0..2,0..2] OF LREAL := ControlParameters.controllerK;
	poseError: RobotPoseSimple;
	vtrans_max: LREAL := ControlParameters.vtrans_max;
	vrot_max: LREAL   := ControlParameters.vrot_max; //vTheta
	u: ARRAY[0..2] OF LREAL;
	i: INT;
	accuracyXY: LREAL := ControlParameters.accuracyXY;
	accuracyTheta: LREAL := ControlParameters.accuracyTheta;
END_VAR



//1.) calculate pose errors
poseError.x 	:= xRobotPoseRef.x 		- xRobotPose.x;
poseError.y 	:= xRobotPoseRef.y 		- xRobotPose.y;
poseError.theta := xRobotPoseRef.theta 	- xRobotPose.theta;

reachedReference := (ABS(poseError.x) < accuracyXY) AND (ABS(poseError.y) < accuracyXY) AND (ABS(poseError.theta) < accuracyTheta);

//2.) apply gain on errors
FOR i := 0 TO 2 DO
	u[i] := K[0,i] * poseError.x + K[1,i] * poseError.y + K[2,i] * poseError.theta;
END_FOR;

//3.) apply saturation
FOR i := 0 TO 1 DO
	IF u[i] > vtrans_max THEN
		u[i] := vtrans_max;
	ELSIF u[i] < -vtrans_max THEN
		u[i] := -vtrans_max;
	END_IF
END_FOR

IF u[2] > vrot_max THEN
	u[2] := vrot_max;
ELSIF u[2] < -vrot_max THEN
	u[2] := -vrot_max;
END_IF

//4.) set control outputs
IF enable THEN
	vXrobot 	:= (u[0] + xRobotvelRef.x);
	vYrobot 	:= (u[1] + xRobotvelRef.y);
	omegaRobot	:= (u[2] + xRobotvelRef.theta);
ELSE
	vXrobot 	:= 0;
	vYrobot 	:= 0;
	omegaRobot  := 0;
END_IF

METHOD reset : BOOL
VAR_INPUT
END_VAR
reachedReference := FALSE;
reset := TRUE;
END_METHOD

END_FUNCTION_BLOCK

// ---- POUs/UserPOUs/GW3ControlAlgorithm/TimeOptimalTrajectory.TcPOU
FUNCTION_BLOCK TimeOptimalTrajectory
VAR_INPUT
	currentPose			: RobotPoseSimple;
	drive				: BOOL 				:= FALSE;
END_VAR
VAR_OUTPUT
	finished			: BOOL 				:= FALSE;
	ready				: BOOL				:= FALSE;
	generationFailed	: BOOL				:= FALSE;
	pathReady			: BOOL				:= FALSE;
	referencePose		: RobotPoseSimple;
	referenceVelocities	: RobotPoseSimple;
	WPLidx 				: INT 				:= 0;
	path				: Path;
END_VAR
VAR
	trajectoryPlanner	: TrajectoryPlanner;
	wayPointListRaw		: ARRAY [0..100] OF RobotPoseSimple;
	cnt					: INT 				:= 0;
	
    maxRadius		    : LREAL				:= ControlParameters.maxRadius;
	
	samplingTime		: LREAL				:= ControlParameters.samplingTime;
	
	maxVel				: LREAL				:= ControlParameters.maxVel;
	maxAcc				: LREAL				:= ControlParameters.maxAcc;
	
	arcLengthSlow		: LREAL				:= ControlParameters.arcLengthSlow;
	maxSlowVel			: LREAL				:= ControlParameters.maxSlowVel;
	
	maxRotVel			: LREAL				:= ControlParameters.maxRotVel;
	maxRotAcc			: LREAL				:= ControlParameters.maxRotAcc;	
	
	thetaDZ				: LREAL				:= ControlParameters.thetaDZ;
END_VAR

ready 				:= trajectoryPlanner.trajectoriesReady;
generationFailed	:= trajectoryPlanner.trajectoryGenerationFailed;
pathReady 			:= path.ready;

IF cnt = LREAL_TO_INT(samplingTime/Var_HAWIno.CONTROLLER_CYCLE_TIME) AND NOT finished THEN
	WPLidx := WPLidx +1;
	cnt := 0;
END_IF

IF  trajectoryPlanner.posTrajectory[WPLidx].x = -1 AND trajectoryPlanner.posTrajectory[WPLidx].y = -1  AND trajectoryPlanner.posTrajectory[WPLidx].theta = -1 THEN
	finished := TRUE;
END_IF

IF drive AND NOT finished AND ready THEN
	referencePose := trajectoryPlanner.posTrajectory[WPLidx];
	referenceVelocities := trajectoryPlanner.velTrajectory[WPLidx];
	cnt := cnt +1;	
END_IF

METHOD calculateTrajectoryContraints : BOOL
VAR_INPUT
END_VAR
VAR
	rotationPerArcLength: LREAL;
	mVel, mAcc, bVel, bAcc: LREAL;
	endPoint, startPoint: RobotPoseSimple;
END_VAR
maxVel  := ControlParameters.maxVel;
maxAcc	:= ControlParameters.maxAcc;
IF path.length-2*ControlParameters.thetaDZ > 0 THEN
	endPoint := path.endPointVal;
	startPoint :=  path.startPointVal;
	rotationPerArcLength := ABS((endpoint.theta-startPoint.theta)/(path.length-2*ControlParameters.thetaDZ));
	IF rotationPerArcLength >= pi/(1-2*ControlParameters.thetaDZ) THEN
		maxVel  := 0.3;
		maxAcc	:= 0.2;
	ELSIF rotationPerArcLength > pi/(1.5-2*ControlParameters.thetaDZ) AND  rotationPerArcLength < pi/(1-2*ControlParameters.thetaDZ) THEN
		mVel :=  (0.3-ControlParameters.maxVel)/(pi/(1-2*ControlParameters.thetaDZ- pi/(1.5-2*ControlParameters.thetaDZ)));
		bVel := ControlParameters.maxVel-mVel*pi/1.1;
		mAcc :=  (0.2-ControlParameters.maxAcc)/(pi/(1-2*ControlParameters.thetaDZ- pi/(1.5-2*ControlParameters.thetaDZ)));
		bAcc := ControlParameters.maxAcc-mAcc*pi/1.1;
		maxVel := mVel*rotationPerArcLength + bVel;
		maxAcc := mAcc*rotationPerArcLength + bAcc;
	END_IF
END_IF
END_METHOD

METHOD generateTrajectory : BOOL
VAR_INPUT
END_VAR
trajectoryPlanner.generateTrajectory();
END_METHOD

METHOD reset : BOOL
VAR_INPUT
END_VAR
WPLidx 			:= 0; 						//reset
finished 		:= FALSE;

path.reset();
trajectoryPlanner.reset();
reset := TRUE;
END_METHOD

METHOD setRobotPose : RobotPoseSimple
VAR_INPUT
	newPose: RobotPoseSimple;
END_VAR
//not needed here
END_METHOD

METHOD setWaypointList : ARRAY [0..100] OF RobotPoseSimple
VAR_INPUT
	newWayPointList	: ARRAY [0..100]  OF RobotPoseSimple;
END_VAR

VAR
	extendedWayPointList			:	ARRAY [0..101] OF RobotPoseSimple;
	i								: INT;
	maxInitialPoseError				: LREAL := 50;		// unit: mm
END_VAR
// Insert actual position as first waypoint if robot is too far away from first
// x and y have to be < 100 => noise of encoder integrates onto invalid cam data, (100,100) is still an invalid point
IF (SQRT(EXPT(currentPose.x - newWayPointList[0].x, 2) + EXPT(currentPose.y - newWayPointList[0].y, 2)) > maxInitialPoseError) AND currentPose.x > 100 AND currentPose.y > 100  THEN
	// shift all elements +1 to right except the lat one (gets overwritten)
	FOR i := 100 TO 0 BY -1 DO
		extendedWayPointList[i + 1] := newWayPointList[i];
	END_FOR

	// insert actual pose as first waypoint
	extendedWayPointList[0] := currentPose;
ELSIF newWayPointList[1].x = -1 AND newWayPointList[1].y = -1 THEN //only one point in wpl
	extendedWayPointList[0] := currentPose;
	extendedWayPointList[1] := newWayPointList[0];
	extendedWayPointList[2] := newWayPointList[1]; //(-1, -1, -1)
ELSE
	//dont shift all elements
	FOR i := 0 TO 100 BY 1 DO
		extendedWayPointList[i] := newWayPointList[i];
	END_FOR
	
	extendedWayPointList[101].x := -1;
	extendedWayPointList[101].y := -1;
	extendedWayPointList[0].theta := currentPose.theta;
END_IF

path(waypointListRaw := extendedWayPointList, maxRadius := maxRadius, thetaDZ := thetaDZ);



IF path.ready THEN
	calculateTrajectoryContraints();	//zur Not auskommentieren
	trajectoryPlanner(path := path, 
				  qAccMax := maxAcc, 
				  qVelMax := maxVel, 
				  thetaAccMax := maxRotAcc,
				  thetaVelMax := maxRotVel,
				  qVelMaxSlow := maxSlowVel,
				  arcLengthSlow := arcLengthSlow,
				  deltaT := samplingTime);
 END_IF
END_METHOD

END_FUNCTION_BLOCK

// ---- POUs/UserPOUs/GW3PathAndTrajectoryPlanning/Path.TcPOU
FUNCTION_BLOCK Path EXTENDS Spline
VAR_INPUT
	waypointListRaw: 	ARRAY [0..101] OF RobotPoseSimple;
	maxRadius: 			LREAL;
	thetaDZ: 			LREAL := 0.1;
END_VAR
VAR_OUTPUT
	ready: 				BOOL;
END_VAR
VAR
	waypointList: 		ARRAY [0..101] 	OF 	RobotPoseSimple;
		
	subsplines: 		ARRAY [0..100] 	OF  POINTER TO Spline;
	linearSplines:		ARRAY [0..51] OF LinearSpline;
	bezierCurves:		ARRAY [0..49] OF BezierCurve;
	
	transitions: 		ARRAY [0..100] 	OF LREAL;
	nmbOfSubsplines, nmbOfPreprocessedWaypoints: INT;
	subsplineGenerationIdx:						 INT := 1;
	generatedSubsplines:						 BOOL := FALSE;
END_VAR

IF NOT generatedSubsplines THEN
	preprocessWaypointlist();
	nmbOfSubsplines := 2*nmbOfPreprocessedWaypoints-3;
	generateSubsplines();	
END_IF

IF generatedSubsplines AND NOT ready THEN
	lengthVar := calculateLength();
	calculateTransitions();
	
	startPoint := subsplines[0]^.startPointVal;
	endPoint   := subsplines[nmbOfSubsplines-1]^.endPointVal;
	
	startPoint.theta := waypointList[0].theta;
	
	endPoint.theta	 := waypointList[nmbOfPreprocessedWaypoints-1].theta;
	IF ABS(endPoint.theta-startPoint.theta) > ABS(endPoint.theta+2*pi-startPoint.theta) THEN
		endPoint.theta := endPoint.theta+2*pi;
	ELSIF ABS(endPoint.theta-startPoint.theta) > ABS(endPoint.theta-2*pi-startPoint.theta) THEN
		endPoint.theta := endPoint.theta-2*pi;
	END_IF
	
	ready := TRUE;
END_IF

(* 
Implementation of abstract Spline method.
For internal inital length calculation, should be called in the constructor => protected
*)
METHOD PROTECTED  calculateLength : LREAL
VAR_INPUT
END_VAR
VAR
	i: INT;
END_VAR
calculateLength := 0;
FOR i := 0 TO nmbOfSubsplines-1 DO
	calculateLength := calculateLength + subsplines[i]^.length;
END_FOR
END_METHOD

METHOD PRIVATE calculateTransitions
VAR_INPUT
END_VAR
VAR
	i : INT;
END_VAR
transitions[0] := 0;
FOR i := 0 TO nmbOfSubsplines-2 DO
	transitions[i+1] := transitions[i] + subsplines[i]^.length;
END_FOR
END_METHOD

(* 
Implementation of abstract Spline method.
Calculates the derivate of the spline at an arbitrary arcLength. Should be implmented for order one and two. Invalid 
orders should write a -1 in every component of the return value.
*)
METHOD  PUBLIC diff : RobotPoseSimple
VAR_INPUT
	arcLength: LREAL; //arcLength at which the corresponding derivative should be calculated
	order: INT := 1;  //optional: order of the derivate, should be implemented for 1 and 2, default: 1
END_VAR
VAR
	subspline: 				POINTER TO Spline;
	arcOffset, deltaTheta: 	LREAL;
	dPos: RobotPoseSimple;
END_VAR
getSubsplineToPoint(arcLength := arcLength,
					subspline => subspline,
					arcOffset => arcOffset);
deltaTheta:= endPoint.theta - startPoint.theta; 		
diff 		:= subspline^.diff(arcLength := arcOffset, order:= order);	
diff.theta 	:= dTheta(arcLength := arcLength, order := order);
END_METHOD

METHOD PRIVATE dTheta : LREAL
VAR_INPUT
	arcLength: LREAL;
	order: INT;
END_VAR
VAR
	deltaTheta: LREAL;
END_VAR
deltaTheta := endPoint.theta - startPoint.theta;
IF arcLength < thetaDZ  OR arcLength > lengthVar - thetaDZ THEN
	dTheta := 0;
ELSIF order = 1 THEN
	dTheta := deltaTheta/2*(pi/(lengthVar-2*thetaDZ))*SIN(pi/(lengthVar-2*thetaDZ)*(arcLength-thetaDZ));
ELSIF order = 2 THEN
	dTheta := deltaTheta/2*EXPT(pi/(lengthVar-2*thetaDZ),2)*COS(pi/(lengthVar-2*thetaDZ)*(arcLength-thetaDZ));
END_IF
END_METHOD

METHOD generateSubsplines : BOOL
VAR_INPUT
END_VAR
VAR

			
	//xTmpLinear,yTmpLinear:    		ARRAY [0..1] OF LREAL;
	wplTmpLinear:					ARRAY [0..1] OF RobotPoseSimple;
	//xTmpBezier,yTmpBezier:    		ARRAY [0..2] OF LREAL;
	wplTmpBezier:					ARRAY [0..2] OF RobotPoseSimple;
	
	i,j,k: INT := 0;
END_VAR
IF nmbOfSubsplines <> 1 AND NOT ready THEN 
	IF subsplineGenerationIdx = 0 THEN
		//first Segment is always linear
		wplTmpLinear[0] := waypointList[0];
		wplTmpLinear[1] := subsplines[1]^.startPointVal;
		linearSplines[0](wayPoints := wplTmpLinear);
		subsplines[0] := ADR(linearSplines[0]);
		subsplineGenerationIdx := nmbOfSubsplines-1;
	ELSIF subsplineGenerationIdx = nmbOfSubsplines-1 THEN
		//last Segment is always linear
		wplTmpLinear[0] := subsplines[nmbOfSubsplines-2]^.endPointVal;
		wplTmpLinear[1] := waypointList[nmbOfPreprocessedWaypoints-1];
		linearSplines[(nmbOfSubsplines+1)/2](wayPoints := wplTmpLinear);
		subsplines[nmbOfSubsplines-1] := ADR(linearSplines[(nmbOfSubsplines+1)/2]);
		IF nmbOfSubsplines = 3 THEN
			generatedSubsplines := TRUE; //if only three subsplines path geenreation stops here
		ELSE
			subsplineGenerationIdx := 2; //if more then three subsplines then go on
		END_IF
	ELSIF (subsplineGenerationIdx MOD 2) <> 0 THEN
		i := subsplineGenerationIdx;
		k := 0;
		
		//extract relevant points for bezier curve creation
		FOR j := (i-1)/2 TO (i-1)/2+2 BY 1 DO
			wplTmpBezier[k] := waypointList[j];
			k := k + 1;
		END_FOR
  
		bezierCurves[(i-1)/2](waypoints:=wplTmpBezier, maxRadius := maxRadius);
		subsplines[i]:= ADR(bezierCurves[(i-1)/2]);
		
		IF subsplineGenerationIdx >= nmbOfSubsplines-2 THEN
			subsplineGenerationIdx := 0;
		ELSE 
			subsplineGenerationIdx := i+2;
		END_IF
	ELSIF (subsplineGenerationIdx MOD 2) = 0 THEN
		i := subsplineGenerationIdx;
		wplTmpLinear[0] := subsplines[i-1]^.endPointVal;
		wplTmpLinear[1] := subsplines[i+1]^.startPointVal;
		linearSplines[i/2](wayPoints := wplTmpLinear);
		subsplines[i] := ADR(linearSplines[i/2]);
		IF subsplineGenerationIdx >= nmbOfSubsplines-3 THEN
			generatedSubsplines := TRUE;
		ELSE	
		subsplineGenerationIdx := subsplineGenerationIdx + 2;
		END_IF
	END_IF
ELSIF nmbOfSubsplines = 1 AND NOT ready THEN  //nmbOfSubsplines = 1  => only one linear Segment
	wplTmpLinear[0] := waypointList[0];
	wplTmpLinear[1] := waypointList[1];;
	linearSplines[0](wayPoints := wplTmpLinear);
	subsplines[0] := ADR(linearSplines[0]);
	generatedSubsplines := TRUE;
END_IF
END_METHOD

(*
Implementation of abstract Spline method.
Gets the configuration of the Spline at any given arcLength. 
*)
METHOD PUBLIC  getPoint : RobotPoseSimple
VAR_INPUT
	arcLength: LREAL; //arcLength at which the Splines configuration shall be calculated.
END_VAR
VAR
	subspline: POINTER TO Spline;
	arcOffset: LREAL;
	deltaTheta: LREAL;
END_VAR
getSubsplineToPoint(arcLength := arcLength,
					subspline => subspline,
					arcOffset => arcOffset);
getPoint := subspline^.getPoint(arcLength:= arcOffset);

deltaTheta 		:= endPoint.theta - startPoint.theta;
getPoint.theta	:= theta(arcLength := arcLength);
END_METHOD

METHOD PRIVATE getSubsplineToPoint : POINTER TO Spline
VAR_INPUT
	arcLength: LREAL;
END_VAR

VAR_OUTPUT
	subspline: 	POINTER TO Spline;
	arcOffset: 	LREAL;
	i: 			INT := 0;
END_VAR
arcOffset := arcLength;
IF arcLength >= length THEN
	arcOffset := arcLength - transitions[nmbOfSubsplines-1];
	subspline := subsplines[nmbOfSubsplines-1];
	RETURN;
END_IF

FOR i := 0 TO nmbOfSubsplines-1 DO
	IF arcOffset-subsplines[i]^.length < 0 THEN
		subspline := subsplines[i];
		EXIT;
	ELSE
		arcOffset := arcOffset -subsplines[i]^.length;
	END_IF
END_FOR
END_METHOD

METHOD getSwitchingPointIntervals : ARRAY [0..98] OF LREAL
VAR_INPUT
END_VAR
VAR
	i: INT := 0;
END_VAR
FILL(arr :=  getSwitchingPointIntervals, val := -1.0);
FOR i := 1 TO nmbOfSubsplines-1 BY 1 DO
	getSwitchingPointIntervals[i-1] := transitions[i];
END_FOR
END_METHOD

METHOD PRIVATE preprocessWaypointlist 
VAR_IN_OUT
END_VAR
VAR 
	i : 				INT 			:= 0;
	nextIDX: 			INT;
	phi1, phi2: 		LREAL;
	alpha1, alpha2: 	LREAL;
END_VAR
waypointList[0].theta := waypointListRaw[0].theta;	
waypointList[0].y := waypointListRaw[0].y/1000;	
waypointList[0].x := waypointListRaw[0].x/1000;	
nextIDX := 1;

FOR i := 1 TO 99 DO
	//exit if last point is reached, last valid point is last point in preprocessed list
	IF waypointListRaw[i+1].x = -1 AND waypointListRaw[i+1].y = -1 THEN
		waypointList[nextIDX].theta := waypointListRaw[i].theta;	
		waypointList[nextIDX].y := waypointListRaw[i].y/1000;	
		waypointList[nextIDX].x := waypointListRaw[i].x/1000;	
		EXIT;
	END_IF	

	phi1 := ATAN2(waypointListRaw[i].y-waypointListRaw[i-1].y,waypointListRaw[i].x-waypointListRaw[i-1].x);
	phi2 := ATAN2(waypointListRaw[i+1].y-waypointListRaw[i].y,waypointListRaw[i+1].x-waypointListRaw[i].x);
	alpha1 := phi1;
	alpha2 := phi2;
	
	//alpha1 := normalizeAngle(alpha1, pi, -pi);
	//alpha2 := normalizeAngle(alpha2, pi, -pi);
		
	alpha1 := phi1;
	alpha2 := normalizeAngle(phi2,alpha1+pi,alpha1-pi);
	IF phi1 <> phi2 AND phi1 <> normalizeAngle(phi2, pi, -pi) AND alpha2 <= alpha1+pi/2*1.1 AND alpha2 >= alpha1-pi/2*1.1 THEN
		waypointList[nextIDX].theta := waypointListRaw[i].theta;	
		waypointList[nextIDX].y := waypointListRaw[i].y/1000;	
		waypointList[nextIDX].x := waypointListRaw[i].x/1000;	
		nextIDX := nextIDX +1;
	END_IF
END_FOR
nmbOfPreprocessedWaypoints := nextIDX +1;
END_METHOD

METHOD reset : LREAL
VAR_INPUT
END_VAR
VAR
	i: INT;
END_VAR
startPoint.x 	:= 0;
startPoint.y	:= 0;
startPoint.theta:= 0;

endPoint.x 	:= 0;
endPoint.y	:= 0;
endPoint.theta:= 0;

FOR i := 0 TO nmbOfSubsplines-1 DO
	subsplines[i] := 0;
END_FOR

generatedSubsplines := FALSE;
ready := FALSE;
subsplineGenerationIdx := 1;
END_METHOD

METHOD PRIVATE theta : LREAL
VAR_INPUT
	arcLength: LREAL;
END_VAR
VAR
	deltaTheta: LREAL;
END_VAR
deltaTheta := endPoint.theta - startPoint.theta;
IF arcLength < thetaDZ THEN
	theta := startPoint.theta;
ELSIF arcLength > lengthVar - thetaDZ THEN
	theta := endPoint.theta;
ELSE
	theta := startPoint.theta + deltaTheta/2*(1-COS(pi/(lengthVar-2*thetaDZ)*(arcLength-thetaDZ)));
END_IF
END_METHOD

END_FUNCTION_BLOCK

// ---- POUs/UserPOUs/GW3PathAndTrajectoryPlanning/BezierCurve.TcPOU
(* Class: BezierCurve
This class implements a quadratic BezierCurve. A quadratic BezierCurve is uniquely defined by three Points. In this 
specific application the three points are generated from three Waypoints, a previous, the corner, and the next Waypoint. The corner
Point is directly used as controlPoint. From the prev and nex Wapoints the start and endPoints are generated by intersection of Linear 

*)
FUNCTION_BLOCK BezierCurve EXTENDS Curve
VAR_INPUT
	waypoints: ARRAY[0..2] OF RobotPoseSimple;
	deltaT: LREAL := 1E-3; //only for inital length calculation
	maxRadius : LREAL;		// Max. radius of bezier curves
END_VAR
VAR_OUTPUT
END_VAR
VAR
	prevWP, nextWP, controlPoint	: RobotPoseSimple;
	a2, a1, a0, b2, b1, b0			: LREAL;
	radius							: LREAL := 0.1;				// Calculated radius of bezier curves.
	d1, d2, d						: LREAL;					// Distances to determine radius of bezier curves
END_VAR

controlPoint := waypoints[1];
prevWP := waypoints[0];
nextWP := waypoints[2];

// Compute minimum required radius
d1 := SQRT(EXPT(controlPoint.x - prevWP.x, 2) + EXPT(controlPoint.y - prevWP.y, 2)) - 1E-3;
d2 := SQRT(EXPT(controlPoint.x - nextWP.x, 2) + EXPT(controlPoint.y - nextWP.y, 2)) - 1E-3;
radius := MIN(d1/2, d2/2, maxRadius);

getStartEndPoint();

calculateCoefficients();
lengthVar := calculateLength();

METHOD PRIVATE calculateCoefficients 
VAR_INPUT
END_VAR
a2 := (startPoint.x - 2*controlPoint.x + endPoint.x);
a1 := (2*controlPoint.x - 2*startPoint.x);
a0 := startPoint.x;

b2 := (startPoint.y - 2*controlPoint.y + endPoint.y);
b1 := (2*controlPoint.y - 2*startPoint.y);
b0 := startPoint.y;
END_METHOD

(* 
Implementation of abstract Spline method.
For internal inital length calculation, should be called in the constructor => protected
*)
METHOD PROTECTED  calculateLength : LREAL
VAR_INPUT
END_VAR

VAR
	i : INT;
	t : LREAL;
END_VAR
calculateLength := 0;
FOR i := 0 TO LREAL_TO_INT(1/deltaT)-1 DO
	t := i*deltaT;
	calculateLength := calculateLength + ds(t)*deltaT;
END_FOR
END_METHOD

METHOD PRIVATE dds : LREAL
VAR_INPUT
	t, dsVal: LREAL;
END_VAR
dds := (4*(EXPT(a2,2)+EXPT(b2,2))*t + 2*(a2*a1+b2*b1))/dsVal;
END_METHOD

(* 
Implementation of abstract Spline method.
Calculates the derivate of the spline at an arbitrary arcLength. Should be implmented for order one and two. Invalid 
orders should write a -1 in every component of the return value.
*)
METHOD PUBLIC diff : RobotPoseSimple
VAR_INPUT
	arcLength: LREAL; //arcLength at which the corresponding derivative should be calculated
	order: INT := 1;  //optional: order of the derivate, should be implemented for 1 and 2, default: 1
END_VAR
VAR
	t, dsVal, ddsVal: LREAL;
	dPos, ddPos: RobotPoseSimple;
END_VAR
t 		:= normalize(arcLength);
dPos	:= diffNorm(t);
dsVal 		:= ds(t);
diff.theta := -1;

CASE order OF
	1 :
		diff.x := dPos.x/dsVal;
		diff.y := dPos.y/dsVal;
	2 :
	   //calculate first derivative
	   //inner derivative
		ddsVal := dds(t, dsVal);
		ddPos  := diff2Norm(t);
		
		//calculate second derivate, derivation NOT trivial
		diff.x := ddPos.x*EXPT(dsVal,-2) - dPos.x*EXPT(dsVal, -3) *ddsVal;
		diff.y := ddPos.y*EXPT(dsVal,-2) - dPos.y*EXPT(dsVal, -3) *ddsVal;

ELSE
	diff.x := -1.0;
	diff.y := -1.0;
	diff.theta := -1.0;
END_CASE;
END_METHOD

METHOD PRIVATE diff2Norm : RobotPoseSimple
VAR_INPUT
	t: LREAL;
END_VAR
diff2Norm.x 		:= 2*a2;
diff2Norm.y 		:= 2*b2;
diff2Norm.theta		:= -1; //unused
END_METHOD

METHOD PRIVATE diffNorm : RobotPoseSimple
VAR_INPUT
	t: LREAL;
END_VAR
diffNorm.x := 2*a2*t + a1;
diffNorm.y := 2*b2*t + b1;
END_METHOD

METHOD PRIVATE ds : LREAL
VAR_INPUT
	t: LREAL;
END_VAR
VAR
	dPos: RobotPoseSimple; //first order derivative of BezierCurve after t
END_VAR
dPos := diffNorm(t);
ds := sqrt(EXPT(dPos.x,2) + EXPT(dPos.y,2));
END_METHOD

(*
Implementation of abstract Spline method.
Gets the configuration of the Spline at any given arcLength. 
*)
METHOD PUBLIC getPoint : RobotPoseSimple
VAR_INPUT
	arcLength: LREAL; //arcLength at which the Splines configuration shall be calculated. 
END_VAR

VAR
	t: LREAL;
END_VAR
t := normalize(arcLength);
getPoint := getPointNorm(t);
END_METHOD

METHOD PRIVATE getPointNorm : RobotPoseSimple
VAR_INPUT
	t: LREAL;
END_VAR
getPointNorm.x   := a2*EXPT(t,2) + a1* t + a0;
getPointNorm.y   := b2*EXPT(t,2) +b1 * t + b0;
getPointNorm.theta := -1; //unused
END_METHOD

METHOD PRIVATE getStartEndPoint : RobotPoseSimple
VAR_INPUT
END_VAR

VAR
	phi1, zpx11, zpx12, zpy11, zpy12, zpx1, zpy1: LREAL;
	phi2, zpx21, zpx22, zpy21, zpy22, zpx2, zpy2: LREAL;
END_VAR
//Start point:
// - angle of incidence of former linear part
phi1 := ATAN2(prevWP.y - controlPoint.y, prevWP.x - controlPoint.x);

// - x-coordinates where former linear part intersects with circle
zpx11 := controlPoint.x - radius*COS(phi1);
zpx12 := controlPoint.x + radius*COS(phi1);

//- y-coordinates where former linear part intersects with circle
zpy11 := controlPoint.y - radius*SIN(phi1);
zpy12 := controlPoint.y + radius*SIN(phi1);

//- decide which of the 2 solutions the relevant one
//(left or right intersection)
IF prevWP.x < controlPoint.x THEN
	zpx1 := MIN(zpx11, zpx12);
ELSE
	zpx1 := MAX(zpx11, zpx12);
END_IF

//- decide which of the 2 solutions the relevant one
//(left or right intersection)
IF prevWP.y < controlPoint.y THEN
	zpy1 := MIN(zpy11, zpy12);
ELSE
	zpy1 := MAX(zpy11, zpy12);
END_IF

//ZP 2:
//- angle of incidence of following linear part
phi2 := atan2(nextWP.y - controlPoint.y, nextWP.x - controlPoint.x);

// - x-coordinates where following linear part intersects with circle
zpx21 := controlPoint.x - radius*COS(phi2);
zpx22 := controlPoint.x + radius*COS(phi2);

//- y-coordinates where former linear part intersects with circle
zpy21 := controlPoint.y - radius * SIN(phi2);
zpy22 := controlPoint.y + radius * SIN(phi2);

// - decide which OF the 2 solutions the relevant one
// (left or right intersection)
IF nextWP.x < controlPoint.x THEN
	zpx2 := MIN(zpx21, zpx22);
else
	zpx2 := MAX(zpx21, zpx22); 
END_IF

IF nextWP.y < controlPoint.y THEN
	zpy2 := MIN(zpy21, zpy22);
else
	zpy2 := MAX(zpy21, zpy22);
END_IF


startPoint.x := zpx1;
startPoint.y := zpy1;
startPoint.theta := phi1;
endPoint.x := zpx2;
endPoint.y := zpy2;
endPoint.theta := phi2;
END_METHOD

METHOD PRIVATE normalize : LREAL
VAR_INPUT
	arcLength: LREAL; //corresponds to 's' in MATLAB
END_VAR

VAR
	t_prev: LREAL;
	tol: LREAL := 1E-3;
	i: INT := 0;
	t: LREAL;
END_VAR
t_prev := 2;
WHILE ABS(t-t_prev) > tol AND i < 100 DO
	t_prev := t;
	t := t - (tToArcLength(t) - arcLength) / ds(t);
	i := i +1;
END_WHILE
normalize := t;
END_METHOD

METHOD PRIVATE tToArcLength : LREAL //s(t), corresponds to MATLAB method s in BezierCurve
VAR_INPUT
	t: LREAL;
END_VAR
VAR
	It, I0: LREAL;
END_VAR
tToArcLength := tToArcLengthIntegral(t) - tToArcLengthIntegral(0);
END_METHOD

METHOD PRIVATE tToArcLengthIntegral : LREAL
VAR_INPUT
	t: LREAL;
END_VAR
VAR
	z1,z2,z3,z4,z5,z6:LREAL;
END_VAR
z2 :=4*a2*a1+4*b1*b2;
z3 := 4*EXPT(a2,2)+4*EXPT(b2,2);
z6 := EXPT(a1,2)+EXPT(b1,2);
z1 := t*z2+z6+EXPT(t,2)*z3;
z4 :=(z2/2+t*z3)/SQRT(z3)+ SQRT((t*z2+z6+EXPT(t,2)*z3));
z5 := LN(z4);
tToArcLengthIntegral := (t/2 + z2 / (4*z3)) * SQRT(z1) - (z5* ((EXPT(z2,2) / 4-z3*z6))) / (2*SQRT(EXPT(z3,3) ));
END_METHOD

END_FUNCTION_BLOCK

// ---- POUs/UserPOUs/GW3PathAndTrajectoryPlanning/Curve.TcPOU
(*Class Curve
This class defines the general Structure and the relevant Methods of a concrete Spline. Since it does not make sense to instantiate
a generalized Spline this class is abstract. Concrete Splines which extend this class have to provide Methods for getting Points to 
a arbitrary arcLength (getPoint), getting first respectively second derivates of itself at an arbitrary arcLength (diff). The generalized 
Properties provided by this class is the length of a Spline. startPoint and an endPoint.
*)
FUNCTION_BLOCK ABSTRACT Curve
VAR_INPUT
END_VAR
VAR_OUTPUT
END_VAR
VAR
	lengthVar     :LREAL;				//length of the Spline
	startPoint 	  : RobotPoseSimple;	//startPoint of the Spline
	endPoint      : RobotPoseSimple;	//endPoint of the Spline
END_VAR

(* 
IMPLEMENTATION IN SUBCLASS
For internal inital length calculation, should be called in the constructor => protected
*)
METHOD PROTECTED ABSTRACT calculateLength : LREAL
VAR_INPUT
END_VAR
END_METHOD

(* 
IMPLEMNTATION IN SUBCLASS 
Calculates the derivate of the spline at an arbitrary arcLength. Should be implmented for order one and two. Invalid 
orders should write a -1 in every component of the return value.
*)
METHOD ABSTRACT diff : RobotPoseSimple
VAR_INPUT
	arcLength: LREAL; //arcLength at which the corresponding derivative should be calculated
	order: INT := 1;  //optional: order of the derivate, should be implemented for 1 and 2, default: 1
END_VAR
END_METHOD

(*endpoint of the spline*)
PROPERTY endPointVal : RobotPoseSimple
GET
endPointVal := endPoint;
END_GET
SET
END_SET
END_PROPERTY

(*
IMPLEMENTATION IN SUBCLASS
Gets the configuration of the Spline at any given arcLength. 
*)
METHOD PUBLIC ABSTRACT getPoint : RobotPoseSimple
VAR_INPUT
	arcLength: LREAL;
END_VAR
END_METHOD

(* Length of the Spline*)
PROPERTY length : LREAL
GET
 length := lengthVar;
END_GET
SET
END_SET
END_PROPERTY

(* Startpoint of the Spline *)
PROPERTY startPointVal : RobotPoseSimple
GET
startPointVal.x := startPoint.x;
startPointVal.y := startPoint.y;
startPointVal.theta := startPoint.theta;
END_GET
SET
END_SET
END_PROPERTY

END_FUNCTION_BLOCK

// ---- POUs/UserPOUs/UserFunctions/FILL.TcPOU
//fills all elements of an array of LREAL with a arbitrarly value 
FUNCTION FILL
VAR_IN_OUT
	arr: ARRAY [*] OF LREAL;
END_VAR
VAR_INPUT
	val: LREAL;
END_VAR
VAR
	i : DINT := 0;
END_VAR

FOR i := LOWER_BOUND(arr,1) TO UPPER_BOUND(arr, 1) BY 1 DO
	arr[i] := val;
END_FOR

END_FUNCTION

// ---- POUs/UserPOUs/GW3PathAndTrajectoryPlanning/TrajectoryPlanner.TcPOU
(*TrajectoryPlanner:
This class implements a Trajectory planning algorithm for time optimal generation of velocity profiles along a two times continous differentiable path. The key idea was taken from the paper "Time-Optimal Trajectory Generation for Path
Following with Bounded Acceleration and Velocity" by Tobias Kunz and Mike Stilman (Georgia Institute of Technology). The approach in the paper was adapted to fit the contraints given from a omni-directional
robot.
TODO: implement Method for VAR_OUTPUT generation after trajectory generation has finished.
*)
FUNCTION_BLOCK TrajectoryPlanner
VAR_INPUT
	path:		 	Path;			//path object for which the trajectory should be generated
	qAccMax: 		LREAL;			//maximum tangential path acceleration
	qVelMax: 		LREAL;			//maximum tangential path velocity
	
	qVelMaxSlow:	LREAL;			//maximum tangential path slow velocity
	arcLengthSlow:	LREAL;			//arcLength from the end of path where the robots max velocity is further restricted to qVelMaxSlow
	
	thetaAccMax: 	LREAL;			//maximum angular acceleration
	thetaVelMax: 	LREAL; 			//maximum angular velocity
	deltaT	   :    LREAL := 0.05;	//optional: sampling time of the velocity in [s], default: 50ms
END_VAR
VAR_OUTPUT
	posTrajectory: 					ARRAY	[0..1000] 	OF RobotPoseSimple;			 	//reference position profile. position in global coordinates pver time
	velTrajectory:					ARRAY	[0..1000] 	OF RobotPoseSimple; 			//reference velocity profile, velocity over time
	trajectoryGenerationFinished:	BOOL 									:= FALSE; 	//TRUE if trajectory generation finished successfully
	trajectoryGenerationFailed: 	BOOL 									:= FALSE; 	//TRUE if trajectory generation failed, most likely because something went wrong while integrating backward
	trajectoriesReady:				BOOL 									:= FALSE; 	//TRUE if the generated path trajectories are transformed back into xy-theta-Coordinates
END_VAR
VAR
	searchTol 	: LREAL := 1E-4;	//tolerance for switching point search, switching points are determined by bisection method
	zeroTol		: LREAL := 1E-10;	//numerical zero tolerance
	diffDelta   : LREAL := 1E-6; 	//dt for calculation of dVelMaxAcc
	currentStep : INT 	:= 1;		//indicates current algorithm step
	
	maxIter				: INT := 100; 				//maximum allowed iterations for while loop of bisection method
	acc					: LREAL;					//acceleration for the next time step in the algorithm
	searchPos			: LREAL;					//position from which the swithing point search starts
	swp					: ARRAY[0..99] OF LREAL;	//array of switching points, not needed entrys are filled with -1
	nmbSWP				: INT;						//number of swichting points
	
	pos			: ARRAY[0..1000] OF LREAL;			//the i-th element indicates the position on the curve at time t=i*deltaT
	vel			: ARRAY[0..1000] OF LREAL;			//the i-th element indicates the tangential path velocity on the curve at time t=i*deltaT
	idxForward  : INT := 0;							//index Variable for writing into pos and vel, i-th element represents t=i*deltaT
	
	posBackward	: ARRAY[0..1000] OF LREAL;			//temp array for backward integrartion, after backward integration is finished the values are written into pos
	velBackward	: ARRAY[0..1000] OF LREAL; 			//temp array for backward integrartion, after backward integration is finished the values are written into vel
	idxBackward : INT := 0;							//temp index Variable for writing into posBackward and velBackward, i-th element indicates time t_bw=i*deltaT since backward integration started

	integratingBWfromPathEnd: 		BOOL := FALSE;	//indicates that the last backward integration process started, needed internally for setting trajectoryGenerationFinished-Flag appropriate
END_VAR

calculateSWP();

METHOD PRIVATE accMax : LREAL
VAR_INPUT
	arcLength: LREAL;
	velocity: LREAL;
END_VAR
VAR
	accMaxSquare: LREAL;
	ddPos: RobotPoseSimple;
END_VAR
ddPos := path.diff(arcLength, 2);

accMaxSquare := EXPT(qAccMax,2)-EXPT(velocity,4)*(EXPT(ddPos.x,2)+EXPT(ddPos.y,2));
IF accMaxSquare > -zeroTol THEN
	accMax := SQRT(ABS(accMaxSquare));
ELSE
	accMax := 0;
END_IF
END_METHOD

METHOD PRIVATE accMin : LREAL
VAR_INPUT
	arcLength: LREAL;
	velocity: LREAL;
END_VAR
accMin := -accMax(arcLength, velocity);
END_METHOD

METHOD PRIVATE calculateSWP : BOOL
VAR_INPUT
END_VAR
VAR
	swpIntervals : ARRAY[0..98] OF LREAL;
	i, k: 	INT;
	maxIdx: INT;
	
	left, right, center, distance: LREAL;
END_VAR
swpIntervals := path.getSwitchingPointIntervals();

//check how many swps there are
FOR i := 0 TO 98 DO
	IF swpIntervals[i] = -1 THEN
		maxIdx := i-1;
		nmbSWP := i/2;
		EXIT;
	END_IF
END_FOR

//find exact SWP by bisection in corresponding interval
FOR i := 0 TO maxIdx BY 2 DO
	left 		:= swpIntervals[i];
	right 		:= swpIntervals[i+1];
	//distance 	:= ABS(right-left);
	
	//improved init because swp is near center of interval
	//left 		:= left+distance/4;
	//right 		:= left-distance/4;
	k := 0;
	WHILE ABS(right-left) > searchTol AND k <= maxIter DO
		center 	:= (left+right)/2;
		IF dVelMaxAcc(left,1)*dVelMaxAcc(center,1) < 0 THEN
			right := center;
		ELSE
			left := center;
		END_IF
		k := k+1;
	END_WHILE
	swp[i/2] := (right+left)/2;
END_FOR

//only add deacceleation swp if path is long enough 
IF path.length > arcLengthSlow+0.1 AND nmbSWP > 0 THEN
	//add last swp at the correct indices for slow deaccelarion at the end
	IF swp[nmbSWP-1] < path.length - arcLengthSlow THEN
		swp[nmbSWP] := path.length - arcLengthSlow;
	ELSE
		FOR i := 0 TO nmbSWP-1 DO
			IF swp[i] > path.length - arcLengthSlow THEN
				FOR k := nmbSWP TO i+1 BY -1 DO
					swp[k] := swp[k-1];
				END_FOR	
				swp[i] := path.length - arcLengthSlow;
				EXIT;
			END_IF
		END_FOR
	END_IF
	nmbSWP := nmbSWP+1;
ELSIF path.length > arcLengthSlow+0.1 AND nmbSWP = 0 THEN
	swp[0] := path.length - arcLengthSlow;
	nmbSWP := 1;
END_IF


//add middle of path for theta-swp
//FOR i := 0 TO nmbSWP-1 DO
//	IF swp[i] > path.length/2 THEN
//		FOR k := nmbSWP TO i+1 BY -1 DO
//			swp[k] := swp[k-1];
//		END_FOR	
//		swp[i] := path.length/2 ;
//		EXIT;
//	END_IF
//END_FOR
//nmbSWP := nmbSWP+1;
END_METHOD

METHOD PRIVATE dVelMaxAcc : LREAL
VAR_INPUT
	arcLength	: LREAL;
	order		: INT 		:= 1;
END_VAR
VAR
	velMaxAccM, velMaxAccP, velMaxAccVal: LREAL;
	dVelMaxAccM, dVelMaxAccP: LREAL;
END_VAR
velMaxAccM := velMaxAcc(arcLength-diffDelta);
velMaxAccP := velMaxAcc(arcLength+diffDelta);
CASE order OF
	1:
		dVelMaxAcc := (velMaxAccP-velMaxAccM)/(2*diffDelta);
	2:
		velMaxAccVal := velMaxAcc(arcLength);
		dVelMaxAccM  := (velMaxAccM-velMaxAccVal)/diffDelta;
		dVelMaxAccP  := (velMaxAccVal-velMaxAccP)/diffDelta;
		dVelMaxAcc := (dVelMaxAccP-dVelMaxAccM)/diffDelta;
END_CASE
END_METHOD

METHOD PRIVATE generateOutputTrajectories
VAR_INPUT
END_VAR
VAR
	i: INT := 0;
	tmpPos, dPos: RobotPoseSimple;
END_VAR
FOR i := 0 TO idxForward-1 BY 1 DO
	tmpPos 					:= path.getPoint(arcLength := pos[i]);
	posTrajectory[i].x		:= tmpPos.x*1000;
	posTrajectory[i].y		:= tmpPos.y*1000;
	posTrajectory[i].theta	:= tmpPos.theta;
	dPos 					:= path.diff(arcLength := pos[i], 1);
	
	velTrajectory[i].x 		:= vel[i]*dPos.x*1000; 
	velTrajectory[i].y  	:= vel[i]*dPos.y*1000;
	velTrajectory[i].theta	:= vel[i]*dPos.theta;
END_FOR

FOR i := idxForward TO 1000  BY 1 DO
	posTrajectory[i].x 		:= -1;
	posTrajectory[i].y		:= -1;
	posTrajectory[i].theta	:= -1;
	velTrajectory[i].x 		:= -1; 
	velTrajectory[i].y  	:= -1;
	velTrajectory[i].theta	:= -1;
END_FOR
END_METHOD

METHOD PUBLIC generateTrajectory : BOOL
VAR_INPUT
END_VAR
IF NOT trajectoryGenerationFinished AND NOT trajectoryGenerationFailed AND idxForward <= 1000 THEN
	CASE currentStep OF
		1:
			step1();
		2:
			step2();
		3:
			step3();
		4:
			step4();
		5:
			step5();
	END_CASE
ELSIF idxForward > 1000 THEN
	trajectoryGenerationFailed := TRUE;
END_IF

IF trajectoryGenerationFinished THEN
	generateOutputTrajectories();
	trajectoriesReady := TRUE;
	trajectoryGenerationFinished := FALSE;
END_IF
END_METHOD

METHOD PUBLIC reset
VAR_INPUT
END_VAR
trajectoryGenerationFailed 		:= FALSE;
trajectoryGenerationFinished 	:= FALSE;
trajectoriesReady 				:= FALSE;

zeros(pos);
zeros(posBackward);
zeros(vel);
zeros(velBackward);
zeros(swp);

nmbSWP		:= 0;
idxForward 	:= 0;
idxBackward := 0;
currentStep := 1;
END_METHOD

//initilize algorithm
METHOD PRIVATE step1 : BOOL
VAR_INPUT
END_VAR
vel[0] 	:= 0;
pos[0] 	:= 0;
acc 	:= accMax(0,0);

idxForward 		:= 1;
currentStep		:= 2;
END_METHOD

//integrate forward until a limit curve is hit
METHOD PRIVATE step2 : BOOL
VAR_INPUT
END_VAR
VAR
	currVelMax, currVelMaxAcc: LREAL;
END_VAR
//calculate new positions and velocities, integrate
//TODO: check if more advanced numerical integration is needed, ATM: euler1
pos[idxForward] := pos[idxForward-1] + vel[idxForward-1]*deltaT;
vel[idxForward] := vel[idxForward-1] + acc*deltaT;

//set acceleration for the new time step
acc := accMax(pos[idxForward], vel[idxForward]);

//transitions
currVelMax 		:= velMax(pos[idxForward]);
currVelMaxAcc	:= velMaxAcc(pos[idxForward]);
IF pos[idxForward] > path.length THEN
	//crossed end of path
	zeros(arr := posBackward);
	zeros(arr := velBackward);
	
	//start integrating backward from the end of the path and velocity 0	
	posBackward[0] := path.length;
	velBackward[0] := 0;
	acc := accMin(posBackward[0], velBackward[0]);
	integratingBWfromPathEnd := TRUE;
	
	//integrate backward
	idxBackward := 1;
	currentStep := 5;
ELSIF vel[idxForward] > currVelMax THEN
	//crossed max velocity
	//follow combined limit curve
	currentStep := 3;
ELSIF vel[idxForward] > currVelMaxAcc THEN
	//crossed max velocity caused by acc limit

	searchPos := pos[idxForward-1];
	
	//get next switching point
	currentStep := 4;
ELSE 
	//if no boundaries are crosesd keep integrating forward
	idxForward := idxForward + 1;
END_IF
END_METHOD

//follow limit curve until one of the transitions fire
METHOD PRIVATE step3 : BOOL
VAR_INPUT
END_VAR
VAR
	currVelMax, currVelMaxAcc, currdVelMaxAcc: LREAL;
	currAccMin, currAccMax: LREAL;
END_VAR
//integrate forward, with last valid velocity
pos[idxForward] := pos[idxForward-1] + vel[idxForward-1]*deltaT;

//follow the combined velocity limit curve
currVelMax 		:= velMax(pos[idxForward]);
currVelMaxAcc	:= velMaxAcc(pos[idxForward]);
vel[idxForward] := MIN(currVelMax, currVelMaxAcc);

currAccMin		   := accMin(pos[idxForward], vel[idxForward]);
currAccMax		   := accMax(pos[idxForward], vel[idxForward]);
currdVelMaxAcc 	   := dVelMaxAcc(pos[idxForward],1);

//transitions
IF pos[idxForward] > path.length THEN
	//crossed end of path
	zeros(arr := posBackward);
	zeros(arr := velBackward);
	
	//start integrating backward from the end of the path and velocity 0	
	posBackward[0] := path.length;
	velBackward[0] := 0;
	acc := accMin(posBackward[0], velBackward[0]);
	integratingBWfromPathEnd := TRUE;
	
	//integrate backward
	idxBackward := 1;
	currentStep := 5;
ELSIF currAccMin/vel[idxForward] > currdVelMaxAcc OR (vel[idxForward]-vel[idxForward-1])/ deltaT < -qAccMax THEN
	//search for the next switching point
	searchPos := pos[idxForward-1];
	
	//get next switching point
	currentStep := 4;
ELSIF currAccMax/vel[idxForward] < currdVelMaxAcc THEN
	//start integrating forward with maxAcc in the next timestep
	currentStep := 2;
	idxForward := idxForward + 1;
ELSE
	//keep following the combined velocity limit curve in the next timestep
	idxForward := idxForward + 1;
END_IF
END_METHOD

//search for the next switching point
METHOD PRIVATE step4 : BOOL
VAR_INPUT
END_VAR
VAR
	nextSWP, currVelMax, currVelMaxAcc : LREAL;
	i : INT := 0;
END_VAR
//find next swp
FOR i := 0 TO nmbSWP-1 BY 1 DO
	IF  searchPos-swp[i] < 0 THEN
		nextSWP := swp[i];
		EXIT;
	END_IF
END_FOR

//prepare backward integration
zeros(arr := posBackward);
zeros(arr := velBackward);
idxBackward := 0;

//get inital velocity, pos and acc
posBackward[0] := nextSWP;

currVelMax 		:= velMax(posBackward[0]);
currVelMaxAcc 	:= velMaxAcc(posBackward[0]);
velBackward[0]  := MIN(currVelMax, currVelMaxAcc);

acc := accMin(posBackward[0], velBackward[0]);

//integrate backward from switching point
idxBackward := 1;
currentStep := 5;
END_METHOD

//integrate backward (from swithcing point or path end) until trajectory is crossed
METHOD PRIVATE step5 : BOOL
VAR_INPUT
END_VAR
VAR
	j:				INT 				:= 0;
	cpmIdxForward:	INT 				:= 0;
	currVelMax, currVelMaxAcc: LREAL;
	checkForTrajCrossing: BOOL := FALSE;
END_VAR
//integrate backward
 posBackward[idxBackward] := posBackward[idxBackward-1] - velBackward[idxBackward-1]*deltaT;
velBackward[idxBackward] := velBackward[idxBackward-1] - acc*deltaT;

//get new minimum acceleration
acc := accMin(posBackward[idxBackward], velBackward[idxBackward]);

//check if forward integrated trajectory is crossed and if yes where
IF posBackward[idxBackward] <= pos[idxForward] THEN
	FOR j := idxForward TO 1 BY -1 DO
		//search for the corresponding idx in the forward generated trajectory
		IF	posBackward[idxBackward] > pos[j-1] THEN
			cpmIdxForward := j-1; 
			checkForTrajCrossing := TRUE;
			EXIT;
		END_IF
	END_FOR
END_IF

currVelMax		:= velMax(posBackward[idxBackward]);
currVelMaxAcc	:= velMaxAcc(posBackward[idxBackward]);
//check velocites of the corresponding point on the forward generated trajectry is crossed
// while integrating backward
IF vel[cpmIdxForward] < velBackward[idxBackward] AND checkForTrajCrossing THEN
	//interchange crossed  part of the forward integrated velocities with the 
	//backward integrated trajectory which is below the crossed part
	FOR j := 0 TO idxBackward-1 DO
		vel[cpmIdxForward+j] := velBackward[idxBackward-1-j];
		pos[cpmIdxForward+j] := posBackward[idxBackward-1-j];
	END_FOR
	
	//initlize velocity, acc, and pos for next step
	idxForward 		:= cpmIdxForward+idxBackward-1;
	currVelMax 		:= velMax(pos[idxForward]);
	currVelMaxAcc	:= velMaxAcc(pos[idxForward]);
	acc				:= accMax(pos[idxForward], MIN(currVelMax, currVelMaxAcc));
	
	//integrate forward in the next iteration step
	idxForward 		:= idxForward + 1;
	currentStep 	:= 2;
	
	IF integratingBWfromPathEnd THEN
		integratingBWfromPathEnd 	 := FALSE;
		trajectoryGenerationFinished := TRUE;
	END_IF
ELSIF ABS(currVelMax- velBackward[idxBackward]) < zeroTol OR ABS(currVelMaxAcc-velBackward[idxBackward]) < zeroTol THEN
	trajectoryGenerationFailed := TRUE;
ELSE
	idxBackward := idxBackward + 1;
END_IF
END_METHOD

METHOD PRIVATE velMax : LREAL
VAR_INPUT
	arcLength: LREAL;
END_VAR
VAR
	dPos: RobotPoseSimple;
END_VAR
//if path is short enough take slow end velocity
IF path.length-0.1 <= arcLengthSlow THEN
	qVelMax := qVelMaxSlow;
END_IF


IF arcLength >= path.length-arcLengthSlow THEN
	//slow down at the end
	velMax := qVelMaxSlow;
ELSE
	//max velocity if not at the end of path
	velMax := qVelMax;
END_IF

//max rotational velocity
//dPos := path.diff(arcLength,1);
//IF ABS(dPos.theta) > zeroTol THEN
//	velMax := MIN(velMax, SQRT(thetaVelMax/ABS(dPos.theta)));
//END_IF
END_METHOD

METHOD PRIVATE velMaxAcc : LREAL;
VAR_INPUT
	arcLength: LREAL;
END_VAR
VAR
	ddPos: RobotPoseSimple;
	den: LREAL;
END_VAR
ddPos := path.diff(arcLength:= arcLength, order := 2);

den := EXPT(ddPos.x,2)+EXPT(ddPos.y,2);
IF ABS(den) > zeroTol THEN
	velMaxAcc := MIN(velMax(arcLength), SQRT(qAccMax/SQRT(den)));
ELSE
	velMaxAcc := velMax(arcLength);
END_IF
END_METHOD

END_FUNCTION_BLOCK

// ---- POUs/UserPOUs/UserFunctions/ZEROS.TcPOU
//Fills an array of LREAL of varible length with zeros
FUNCTION ZEROS
VAR_IN_OUT
	arr: ARRAY [*] OF LREAL;
END_VAR

FILL(arr := arr,val := 0.0);

END_FUNCTION

// ---- POUs/UserPOUs/GW3ControlAlgorithm/Robot.TcPOU
//Robot:
//This FB represents the robot and links the control algorithm with the physical I/O of the robot. It is implemented in a separate FB so it is easily interchangeable with
//simulated robot whenever needed. 
FUNCTION_BLOCK Robot
VAR_INPUT
	enable: BOOL;
	vXref, vYref, vThetaRef: LREAL;
END_VAR
VAR_OUTPUT
	vX, vY, vTheta: LREAL;
	sliderGotTriggered: BOOL;
	bumperGotTriggered: BOOL;
END_VAR
VAR
	sliderTrigger:  F_TRIG;
	sldierTON:		TON;	
	bumperTrigger: R_TRIG;
	i1, i2, i3: INT;
	
	i1Raw AT%I*: UINT;
	i2Raw AT%I*: UINT;
	i3Raw AT%I*: UINT;
	
	//inputs to robot
	vXtoRobot 		AT%Q*: LREAL;
	vYtoRobot		AT%Q*: LREAL;
	vThetaToRobot 	AT%Q*: LREAL;
	
	//outputs from robot
	slider 			AT%I*: BOOL;
	bumper			AT%I*: BOOL;
	vel: 	VelocityMeasurement;
END_VAR

vel();

i1 := UINT_TO_INT(i1Raw);
i2 := UINT_TO_INT(i2Raw);
i3 := UINT_TO_INT(i3Raw);

sldierTON(IN := slider, PT := T#200MS); //slider has to be HIGH for at least 250ms
sliderTrigger(CLK := sldierTON.Q, Q => sliderGotTriggered); 

bumperTrigger(CLK := bumper, Q => bumperGotTriggered);

vX 		:= vel.vXRobot;
vY 		:= vel.vYRobot;
vTheta  := vel.vThetaRobot;

//write control outputs to robot if enabled
IF enable = TRUE THEN
			vXtoRobot     := vXref;
			vYtoRobot	  := vYref;
			vThetaToRobot := vThetaRef;
ELSE
			vXtoRobot     := 0;
			vYtoRobot	  := 0;
			vThetaToRobot := 0;
END_IF

END_FUNCTION_BLOCK

// ---- POUs/UserPOUs/GW3ControlAlgorithm/VelocityMeasurement.TcPOU
FUNCTION_BLOCK VelocityMeasurement
VAR_INPUT
END_VAR
VAR_OUTPUT
	vXRobot, vYRobot, vThetaRobot: LREAL;
END_VAR
VAR
	n1MotorRaw AT%I*: UINT;
	n2MotorRaw AT%I*: UINT;
	n3MotorRaw AT%I*: UINT;
	
	v1Wheel, v2Wheel, v3Wheel: LREAL;
	
	g : LREAL 		:= 0.0625; //gear ratio
	rWheel : LREAL  := 40; // wheel radius
	maxMotorVelocity : LREAL := 3600;
END_VAR

v1Wheel := -UINT_TO_INT(n1MotorRaw)/10000.0*maxMotorVelocity/60.0*g*2*pi*rWheel;
v2Wheel := -UINT_TO_INT(n2MotorRaw)/10000.0*maxMotorVelocity/60.0*g*2*pi*rWheel;
v3Wheel := -UINT_TO_INT(n3MotorRaw)/10000.0*maxMotorVelocity/60.0*g*2*pi*rWheel;

vXRobot:=(v3Wheel - v1Wheel) / (2.0 * COS(30.0*PI/180));  		//in mm / s
vYRobot:=(v1Wheel - 2.0 * v2Wheel + v3Wheel) / 3.0;            //in mm / s
vThetaRobot:=(v1Wheel + v2Wheel + v3Wheel) / (3.0 * 135.0);    //in rad / s

END_FUNCTION_BLOCK

// ---- POUs/UserPOUs/UserFunctions/shiftCamAngle.TcPOU
FUNCTION shiftCamAngle : RobotPose
VAR_INPUT
	path: 		Path;
	camData:			RobotPose;
END_VAR
VAR
	thetaMin, thetaMax: LREAL;
	startPoint, endPoint: RobotPoseSimple;
END_VAR

//calculate shifted upper and lower theta bounds depending on the start and end angles of the path
shiftCamAngle.x 	:= camData.x;
shiftCamAngle.y 	:= camData.y;
shiftCamAngle.theta := camData.theta;
shiftCamAngle.e 	:= camData.e;

startPoint := path.startPointVal;
endPoint   := path.endPointVal;

IF startPoint.theta >= endPoint.theta THEN
	thetaMin := startPoint.theta-1.5*pi;
	thetaMax := startPoint.theta+0.5*pi;
ELSIF startPoint.theta < endPoint.theta THEN
	thetaMin := startPoint.theta-0.5*pi;
	thetaMax := startPoint.theta+1.5*pi;
END_IF

//normalize the camera angle within the prior calculated bounds
IF  camData.x <> 0 AND  camData.y <> 0 THEN
	shiftCamAngle.theta := normalizeAngle(camData.theta, thetaMax, thetaMin);
END_IF

END_FUNCTION

// ---- POUs/UserPOUs/UserFunctions/World2Robot.TcPOU
//Transforamtion of world velocities to robot velocities
FUNCTION World2Robot 
VAR_INPUT	
	vx_world: 	 LREAL;
	vy_world: 	 LREAL;
	omega_world: LREAL;
	theta: 		 LREAL;
END_VAR

VAR_OUTPUT
	vx_robot: 	 LREAL;
	vy_robot: 	 LREAL;
	omega_robot: LREAL;
END_VAR

VAR
END_VAR

vx_robot 	:= COS(theta)*vx_world + SIN(theta)* vy_world;
vy_robot	:= -SIN(theta)*vx_world + COS(theta)*vy_world;
omega_robot := omega_world;

END_FUNCTION

// ---- POUs/UserPOUs/GW2/Kollisionserkennung.TcPOU
PROGRAM Kollisionserkennung
VAR
	robotPoseArray AT%I*: ARRAY[1..8] OF RobotPose;
	robotPoseLokal : ARRAY[1..8] OF RobotPose;
	vxRobot AT%I*: LREAL;
	vyRobot AT%I*: LREAL;
	collisionDetected : BOOL := FALSE;
	robotCollision AT%Q* : ARRAY[0..4] OF BOOL;
		
	xRobot, yRobot: LREAL;
	i, j, k, l, m, n, o : INT := 1;
	quadrant, counter : INT := 0;
	noCamera, cameraDown, permanentDown, stateCameraDown  : BOOL := FALSE;
	
	//Bounding Box
	x1Box,y1Box,x2Box,y2Box,x3Box,y3Box,x4Box,y4Box : LREAL; 
	alpha, beta, gamma, diagonal : LREAL := 0.0;
	breite, laenge : INT;
	
	//Timer
	timer :TON;
	timeValue : TIME := T#2S;
END_VAR

 ////////Main function/////////
timer(IN:= noCamera, PT := timeValue); //Roboter darf 2s blind fahren

//suche die Position des passenden Roboters
FOR i := 1 TO 4 BY 1 DO
	IF i = Var_HAWIno.Robot_Number THEN
		xRobot := robotPoseArray[i].x;
		yRobot := robotPoseArray[i].y;
	END_IF
END_FOR

//350mm Durchmesser des Roboters & 130mm Toleranzabstand
breite := 350 + 80; 
laenge := 350 + 80;
diagonal := SQRT(EXPT(breite,2) + EXPT(laenge,2));
IF vyRobot <> 0 AND vxRobot <> 0 THEN
	gamma  := ATAN2(vyRobot,vxRobot); //Drehung des Roboters
END_IF
beta := ATAN(laenge/breite); //Winkel des festen Dreiecks

//Kameradaten verfügbar 
IF xRobot <> 0 AND yRobot <> 0 THEN
	noCamera := FALSE;
	cameraDown := FALSE;
	
	//Zurücksetzen wenn Kameradaten wieder da
	IF stateCameraDown = TRUE THEN
		stateCameraDown := FALSE;
		FOR n:= 0 TO 4 BY 1 DO
			robotCollision[n] := FALSE;
		END_FOR
	END_IF
	
	//Zwischenspeicher der letzten Positionen lokal wenn die Kameradaten nicht ausfallen
	IF robotPoseArray[1].x <> 0 AND robotPoseArray[1].y <> 0 THEN
		robotPoseLokal[1].x := robotPoseArray[1].x;
		robotPoseLokal[1].y := robotPoseArray[1].y;
	END_IF
	IF robotPoseArray[2].x <> 0 AND robotPoseArray[2].y <> 0 THEN
		robotPoseLokal[2].x := robotPoseArray[2].x;
		robotPoseLokal[2].y := robotPoseArray[2].y;
	END_IF
	IF robotPoseArray[3].x <> 0 AND robotPoseArray[3].y <> 0 THEN
		robotPoseLokal[3].x := robotPoseArray[3].x;
		robotPoseLokal[3].y := robotPoseArray[3].y;
	END_IF
	IF robotPoseArray[4].x <> 0 AND robotPoseArray[4].y <> 0 THEN
		robotPoseLokal[4].x := robotPoseArray[4].x;
		robotPoseLokal[4].y := robotPoseArray[4].y;
	END_IF
	
//Kameradaten ausfallen	
ELSE
	noCamera := TRUE;
	cameraDown := TRUE;
	//Kameradaten länger als 2s ausfallen, setzt die Array auf true
	IF timer.Q THEN
		permanentDown := TRUE;
	ELSE
		permanentDown := FALSE;
	END_IF
END_IF

//Kameradaten ausfallen, dann die lokale Position wird zugegriffen
IF cameraDown = TRUE AND permanentDown = FALSE THEN
	xRobot := robotPoseLokal[Var_HAWIno.Robot_Number].x;
	yRobot := robotPoseLokal[Var_HAWIno.Robot_Number].y;
	
//Kameradaten 2s lang ausfallen, ist die gesamte Array robotCollision True und RobotPoseArray = 0
ELSIF cameraDown = TRUE AND permanentDown = TRUE THEN
	xRobot := 0.0;
	yRobot := 0.0;
	FOR o:= 0 TO 4 BY 1 DO
		IF o = 0 THEN
			robotCollision[o] := TRUE;
		ELSE 
			robotCollision[o] := TRUE;
			robotPoseArray[o].x := 0.0;
			robotPoseArray[o].y := 0.0;
			robotPoseArray[o].theta := 0.0;
			robotPoseArray[o].e := 0.0;
		END_IF
	END_FOR
	stateCameraDown := TRUE;
END_IF

//Bounding Box dreht mit der Roboterblickrichtung
IF gamma >= 0 AND gamma < pi/2 THEN //Quadrant 1
	quadrant := 1;
	alpha := pi/2 - gamma; //Winkel des gedrehten Boxes
	x1Box := xRobot + COS(alpha) * breite;
	y1Box := yRobot - SIN(alpha) * breite;
	x2Box := xRobot + SIN(alpha + beta) * diagonal;
	y2Box := yRobot + COS(alpha + beta) * diagonal;
	x3Box := xRobot - COS(alpha + beta) * diagonal;
	y3Box := yRobot + SIN(alpha + beta) * diagonal;
	x4Box := xRobot - COS(alpha) * breite;
	y4Box := yRobot + SIN(alpha) * breite;	
ELSIF gamma >= pi/2 AND gamma <= pi THEN //Quadrant 2
	quadrant := 2;
	alpha := pi - gamma;
	x1Box := xRobot + SIN(alpha) * breite;
	y1Box := yRobot + COS(alpha) * breite;
	x2Box := xRobot - COS(alpha + beta) * diagonal;
	y2Box := yRobot + SIN(alpha + beta) * diagonal;
	x3Box := xRobot - SIN(alpha + beta) * diagonal;
	y3Box := yRobot - COS(alpha + beta) * diagonal;
	x4Box := xRobot - SIN(alpha) * breite;
	y4Box := yRobot - COS(alpha) * breite;
ELSIF gamma > -pi AND gamma < -pi/2 THEN //Quadrant 3
	quadrant := 3;
	alpha := pi + gamma;
	x1Box := xRobot - SIN(alpha) * breite;
	y1Box := yRobot + COS(alpha) * breite;
	x2Box := xRobot - SIN(alpha + beta) * diagonal;
	y2Box := yRobot + COS(alpha + beta) * diagonal;
	x3Box := xRobot - COS(alpha + beta) * diagonal;
	y3Box := yRobot - SIN(alpha + beta) * diagonal;
	x4Box := xRobot + SIN(alpha) * breite;
	y4Box := yRobot - COS(alpha) * breite;	
ELSIF gamma >= -pi/2 AND gamma < 0 THEN //Quadrant 4
	quadrant := 4;
	alpha := gamma + pi/2;
	x1Box := xRobot - COS(alpha) * breite;
	y1Box := yRobot - SIN(alpha) * breite;
	x2Box := xRobot - COS(alpha + beta) * diagonal;
	y2Box := yRobot - SIN(alpha + beta) * diagonal;
	x3Box := xRobot + SIN(alpha + beta) * diagonal;
	y3Box := yRobot - COS(alpha + beta) * diagonal;
	x4Box := xRobot + COS(alpha) * breite;
	y4Box := yRobot + SIN(alpha) * breite;
END_IF

//Erkennt Roboter Kollision in Box?
FOR k := 1 TO 4 BY 1 DO
	IF k <> Var_HAWIno.Robot_Number THEN
		IF quadrant = 1 THEN
			IF robotPoseLokal[k].x < x2Box AND robotPoseLokal[k].x > x4Box AND robotPoseLokal[k].y < y3Box AND robotPoseLokal[k].y > y1Box THEN
				collisionDetected := TRUE;
			ELSE
				collisionDetected := FALSE;
			END_IF
		ELSIF quadrant = 2 THEN
			IF robotPoseLokal[k].x < x1Box AND robotPoseLokal[k].x > x3Box AND robotPoseLokal[k].y < y2Box AND robotPoseLokal[k].y > y4Box THEN
				collisionDetected := TRUE;
			ELSE
				collisionDetected := FALSE;
			END_IF
		ELSIF quadrant = 3 THEN
			IF robotPoseLokal[k].x < x4Box AND robotPoseLokal[k].x > x2Box AND robotPoseLokal[k].y < y1Box AND robotPoseLokal[k].y > y3Box THEN
				collisionDetected := TRUE;
			ELSE
				collisionDetected := FALSE;
			END_IF
		ELSIF quadrant = 4 THEN
			IF robotPoseLokal[k].x < x3Box AND robotPoseLokal[k].x > x1Box AND robotPoseLokal[k].y < y4Box AND robotPoseLokal[k].y > y2Box THEN
				collisionDetected := TRUE;
			ELSE
				collisionDetected := FALSE;
			END_IF
		END_IF
	END_IF
	
	//Kollision erkannt und die beteiligten Robotern werden True gesetzt
	IF collisionDetected = TRUE THEN
		robotCollision[k] := TRUE;
		robotCollision[Var_HAWIno.Robot_Number] := TRUE; 
	ELSIF collisionDetected = FALSE AND k <> Var_HAWIno.Robot_Number THEN
		robotCollision[k] := FALSE;
	END_IF
END_FOR 

//Keine Roboter kollidieren sich, setzt der Roboter zurück
counter := 0;
FOR l := 1 TO 4 BY 1 DO
	IF robotCollision[l] = FALSE THEN
		counter := counter + 1;
	END_IF
END_FOR
IF counter = 3 THEN
	robotCollision[Var_HAWIno.Robot_Number] := FALSE;
END_IF

END_PROGRAM

